LIN {X 0,Y 474.583,Z 139.364,A -85,B 0,C 180,E1 -7443.623,E2 -7443.623} C_VEL
LIN {X 0,Y 474.627,Z 139.367,A -85,B 0,C 180,E1 -7446.642,E2 -7446.642} C_VEL
LIN {X 0,Y 474.635,Z 139.36,A -85,B 0,C 180,E1 -7450.088,E2 -7450.088} C_VEL
LIN {X 0,Y 474.63,Z 139.358,A -85,B 0,C 180,E1 -7451.634,E2 -7451.634} C_VEL
LIN {X 0,Y 473.949,Z 139.45,A -85,B 0,C 180,E1 -7452.343,E2 -7452.343} C_VEL
LIN {X 0,Y 471.1,Z 139.8,A -85,B 0,C 180,E1 -7453.494,E2 -7453.494} C_VEL
LIN {X 0,Y 468.697,Z 140.106,A -85,B 0,C 180,E1 -7454.421,E2 -7454.421} C_VEL
LIN {X 0,Y 467.662,Z 140.228,A -85,B 0,C 180,E1 -7455.138,E2 -7455.138} C_VEL
LIN {X 0,Y 467.575,Z 140.237,A -85,B 0,C 180,E1 -7455.381,E2 -7455.381} C_VEL
LIN {X 0,Y 467.64,Z 140.231,A -85,B 0,C 180,E1 -7457.854,E2 -7457.854} C_VEL
LIN {X 0,Y 467.625,Z 140.231,A -85,B 0,C 180,E1 -7461.356,E2 -7461.356} C_VEL
LIN {X 0,Y 467.692,Z 140.228,A -85,B 0,C 180,E1 -7463.962,E2 -7463.962} C_VEL
LIN {X 0,Y 467.804,Z 140.212,A -85,B 0,C 180,E1 -7467.417,E2 -7467.417} C_VEL
LIN {X 0,Y 467.841,Z 140.213,A -85,B 0,C 180,E1 -7470,E2 -7470} C_VEL
LIN {X 0,Y 467.646,Z 140.35,A -85,B 0,C 180,E1 -7471.049,E2 -7471.049} C_VEL
LIN {X 0,Y 468.659,Z 146.382,A -85,B 0,C 180,E1 -7472.363,E2 -7472.363} C_VEL
LIN {X 0,Y 468.453,Z 159.385,A -85,B 0,C 180,E1 -7475.056,E2 -7475.056} C_VEL
LIN {X 0,Y 471.335,Z 174.004,A -85,B 0,C 180,E1 -7475.401,E2 -7475.401} C_VEL
LIN {X 0,Y 470.568,Z 266.04,A -85,B 0,C 180,E1 -7476.835,E2 -7476.835} C_VEL
LIN {X 0,Y 470.243,Z 278.777,A -85,B 0,C 180,E1 -7477.19,E2 -7477.19} C_VEL
LIN {X 0,Y 469.971,Z 291.673,A -85,B 0,C 180,E1 -7477.735,E2 -7477.735} C_VEL
LIN {X 0,Y 469.608,Z 303.175,A -85,B 0,C 180,E1 -7478.39,E2 -7478.39} C_VEL
LIN {X 0,Y 469.175,Z 313.348,A -85,B 0,C 180,E1 -7479.128,E2 -7479.128} C_VEL
LIN {X 0,Y 468.657,Z 324.539,A -85,B 0,C 180,E1 -7480.149,E2 -7480.149} C_VEL
LIN {X 0,Y 468.147,Z 334.312,A -85,B 0,C 180,E1 -7481.254,E2 -7481.254} C_VEL
LIN {X 0,Y 467.723,Z 342.539,A -85,B 0,C 180,E1 -7482.4,E2 -7482.4} C_VEL
LIN {X 0,Y 467.364,Z 350.081,A -85,B 0,C 180,E1 -7483.7,E2 -7483.7} C_VEL
LIN {X 0,Y 467.052,Z 357.038,A -85,B 0,C 180,E1 -7485.214,E2 -7485.214} C_VEL
LIN {X 0,Y 466.866,Z 361.993,A -85,B 0,C 180,E1 -7486.62,E2 -7486.62} C_VEL
LIN {X 0,Y 466.721,Z 365.558,A -85,B 0,C 180,E1 -7487.974,E2 -7487.974} C_VEL
LIN {X 0,Y 466.61,Z 368.078,A -85,B 0,C 180,E1 -7489.351,E2 -7489.351} C_VEL
LIN {X 0,Y 466.545,Z 369.678,A -85,B 0,C 180,E1 -7490.942,E2 -7490.942} C_VEL
LIN {X 0,Y 466.524,Z 370.029,A -85,B 0,C 180,E1 -7492.124,E2 -7492.124} C_VEL
LIN {X 0,Y 466.578,Z 369.644,A -85,B 0,C 180,E1 -7493.246,E2 -7493.246} C_VEL
LIN {X 0,Y 466.622,Z 367.819,A -85,B 0,C 180,E1 -7494.943,E2 -7494.943} C_VEL
LIN {X 0,Y 466.775,Z 365.039,A -85,B 0,C 180,E1 -7496.37,E2 -7496.37} C_VEL
LIN {X 0,Y 466.957,Z 361.004,A -85,B 0,C 180,E1 -7497.812,E2 -7497.812} C_VEL
LIN {X 0,Y 467.117,Z 355.698,A -85,B 0,C 180,E1 -7499.236,E2 -7499.236} C_VEL
LIN {X 0,Y 467.404,Z 349.728,A -85,B 0,C 180,E1 -7500.496,E2 -7500.496} C_VEL
LIN {X 0,Y 467.742,Z 342.532,A -85,B 0,C 180,E1 -7501.728,E2 -7501.728} C_VEL
LIN {X 0,Y 468.227,Z 333.765,A -85,B 0,C 180,E1 -7502.938,E2 -7502.938} C_VEL
LIN {X 0,Y 468.666,Z 323.643,A -85,B 0,C 180,E1 -7504.07,E2 -7504.07} C_VEL
LIN {X 0,Y 469.176,Z 313.829,A -85,B 0,C 180,E1 -7504.957,E2 -7504.957} C_VEL
LIN {X 0,Y 469.676,Z 302.364,A -85,B 0,C 180,E1 -7505.784,E2 -7505.784} C_VEL
LIN {X 0,Y 470.13,Z 290.08,A -85,B 0,C 180,E1 -7506.463,E2 -7506.463} C_VEL
LIN {X 0,Y 470.434,Z 277.293,A -85,B 0,C 180,E1 -7506.981,E2 -7506.981} C_VEL
LIN {X 0,Y 470.671,Z 264.549,A -85,B 0,C 180,E1 -7507.311,E2 -7507.311} C_VEL
LIN {X 0,Y 471.315,Z 173.329,A -85,B 0,C 180,E1 -7508.736,E2 -7508.736} C_VEL
LIN {X 0,Y 468.55,Z 159.48,A -85,B 0,C 180,E1 -7509.086,E2 -7509.086} C_VEL
LIN {X 0,Y 468.857,Z 147.777,A -85,B 0,C 180,E1 -7511.456,E2 -7511.456} C_VEL
LIN {X 0,Y 467.637,Z 140.236,A -85,B 0,C 180,E1 -7513.07,E2 -7513.07} C_VEL
LIN {X 0,Y 467.573,Z 140.242,A -85,B 0,C 180,E1 -7516.259,E2 -7516.259} C_VEL
LIN {X 0,Y 467.586,Z 140.24,A -85,B 0,C 180,E1 -7518.722,E2 -7518.722} C_VEL
LIN {X 0,Y 467.566,Z 140.248,A -85,B 0,C 180,E1 -7521.957,E2 -7521.957} C_VEL
LIN {X 0,Y 467.562,Z 140.244,A -85,B 0,C 180,E1 -7525.168,E2 -7525.168} C_VEL
LIN {X 0,Y 467.58,Z 140.238,A -85,B 0,C 180,E1 -7528.261,E2 -7528.261} C_VEL
LIN {X 0,Y 467.575,Z 140.243,A -85,B 0,C 180,E1 -7531.251,E2 -7531.251} C_VEL
LIN {X 0,Y 467.609,Z 140.236,A -85,B 0,C 180,E1 -7534.161,E2 -7534.161} C_VEL
LIN {X 0,Y 467.576,Z 140.243,A -85,B 0,C 180,E1 -7536.997,E2 -7536.997} C_VEL
LIN {X 0,Y 467.621,Z 140.234,A -85,B 0,C 180,E1 -7539.778,E2 -7539.778} C_VEL
LIN {X 0,Y 467.595,Z 140.237,A -85,B 0,C 180,E1 -7542.507,E2 -7542.507} C_VEL
LIN {X 0,Y 467.605,Z 140.238,A -85,B 0,C 180,E1 -7545.197,E2 -7545.197} C_VEL
LIN {X 0,Y 467.657,Z 140.227,A -85,B 0,C 180,E1 -7547.855,E2 -7547.855} C_VEL
LIN {X 0,Y 467.67,Z 140.224,A -85,B 0,C 180,E1 -7551.358,E2 -7551.358} C_VEL
LIN {X 0,Y 467.724,Z 140.22,A -85,B 0,C 180,E1 -7553.963,E2 -7553.963} C_VEL
LIN {X 0,Y 467.852,Z 140.201,A -85,B 0,C 180,E1 -7557.418,E2 -7557.418} C_VEL
LIN {X 0,Y 467.88,Z 140.2,A -85,B 0,C 180,E1 -7560.001,E2 -7560.001} C_VEL
LIN {X 0,Y 467.818,Z 140.211,A -85,B 0,C 180,E1 -7562.584,E2 -7562.584} C_VEL
LIN {X 0,Y 467.712,Z 140.219,A -85,B 0,C 180,E1 -7566.038,E2 -7566.038} C_VEL
LIN {X 0,Y 467.66,Z 140.228,A -85,B 0,C 180,E1 -7568.644,E2 -7568.644} C_VEL
LIN {X 0,Y 467.659,Z 140.231,A -85,B 0,C 180,E1 -7572.146,E2 -7572.146} C_VEL
LIN {X 0,Y 467.616,Z 140.236,A -85,B 0,C 180,E1 -7575.696,E2 -7575.696} C_VEL
LIN {X 0,Y 467.617,Z 140.235,A -85,B 0,C 180,E1 -7579.309,E2 -7579.309} C_VEL
LIN {X 0,Y 467.525,Z 140.246,A -85,B 0,C 180,E1 -7582.075,E2 -7582.075} C_VEL
LIN {X 0,Y 467.561,Z 140.24,A -85,B 0,C 180,E1 -7584.89,E2 -7584.89} C_VEL
LIN {X 0,Y 467.541,Z 140.247,A -85,B 0,C 180,E1 -7587.775,E2 -7587.775} C_VEL
LIN {X 0,Y 467.529,Z 140.243,A -85,B 0,C 180,E1 -7591.037,E2 -7591.037} C_VEL
LIN {X 0,Y 467.564,Z 140.237,A -85,B 0,C 180,E1 -7594.238,E2 -7594.238} C_VEL
LIN {X 0,Y 467.512,Z 140.251,A -85,B 0,C 180,E1 -7597.18,E2 -7597.18} C_VEL
LIN {X 0,Y 467.519,Z 140.247,A -85,B 0,C 180,E1 -7600.271,E2 -7600.271} C_VEL
LIN {X 0,Y 467.518,Z 140.25,A -85,B 0,C 180,E1 -7602.569,E2 -7602.569} C_VEL
LIN {X 0,Y 467.564,Z 140.249,A -85,B 0,C 180,E1 -7605.052,E2 -7605.052} C_VEL
LIN {X 0,Y 467.562,Z 140.248,A -85,B 0,C 180,E1 -7608.726,E2 -7608.726} C_VEL
LIN {X 0,Y 467.554,Z 140.243,A -85,B 0,C 180,E1 -7611.954,E2 -7611.954} C_VEL
LIN {X 0,Y 467.557,Z 140.242,A -85,B 0,C 180,E1 -7615.167,E2 -7615.167} C_VEL
LIN {X 0,Y 467.58,Z 140.242,A -85,B 0,C 180,E1 -7618.26,E2 -7618.26} C_VEL
LIN {X 0,Y 467.547,Z 140.245,A -85,B 0,C 180,E1 -7621.248,E2 -7621.248} C_VEL
LIN {X 0,Y 467.602,Z 140.403,A -85,B 0,C 180,E1 -7624.04,E2 -7624.04} C_VEL
LIN {X 0,Y 469.779,Z 151.706,A -85,B 0,C 180,E1 -7626.176,E2 -7626.176} C_VEL
LIN {X 0,Y 469.174,Z 167.509,A -85,B 0,C 180,E1 -7628.93,E2 -7628.93} C_VEL
LIN {X 0,Y 468.445,Z 185.894,A -85,B 0,C 180,E1 -7632.088,E2 -7632.088} C_VEL
LIN {X 0,Y 468.286,Z 190.998,A -85,B 0,C 180,E1 -7632.958,E2 -7632.958} C_VEL
LIN {X 0,Y 471.16,Z 210.073,A -85,B 0,C 180,E1 -7633.369,E2 -7633.369} C_VEL
LIN {X 0,Y 470.551,Z 299.268,A -85,B 0,C 180,E1 -7634.765,E2 -7634.765} C_VEL
LIN {X 0,Y 470.212,Z 311.843,A -85,B 0,C 180,E1 -7635.114,E2 -7635.114} C_VEL
LIN {X 0,Y 469.706,Z 324.813,A -85,B 0,C 180,E1 -7635.652,E2 -7635.652} C_VEL
LIN {X 0,Y 469.186,Z 337.139,A -85,B 0,C 180,E1 -7636.354,E2 -7636.354} C_VEL
LIN {X 0,Y 468.715,Z 347.709,A -85,B 0,C 180,E1 -7637.132,E2 -7637.132} C_VEL
LIN {X 0,Y 468.201,Z 359.257,A -85,B 0,C 180,E1 -7638.199,E2 -7638.199} C_VEL
LIN {X 0,Y 467.748,Z 367.831,A -85,B 0,C 180,E1 -7639.175,E2 -7639.175} C_VEL
LIN {X 0,Y 467.399,Z 375.747,A -85,B 0,C 180,E1 -7640.261,E2 -7640.261} C_VEL
LIN {X 0,Y 467.089,Z 383.481,A -85,B 0,C 180,E1 -7641.564,E2 -7641.564} C_VEL
LIN {X 0,Y 466.831,Z 390.612,A -85,B 0,C 180,E1 -7643.083,E2 -7643.083} C_VEL
LIN {X 0,Y 466.73,Z 395.361,A -85,B 0,C 180,E1 -7644.383,E2 -7644.383} C_VEL
LIN {X 0,Y 466.646,Z 398.989,A -85,B 0,C 180,E1 -7645.682,E2 -7645.682} C_VEL
LIN {X 0,Y 466.69,Z 400.865,A -85,B 0,C 180,E1 -7646.547,E2 -7646.547} C_VEL
LIN {X 0,Y 466.663,Z 402.269,A -85,B 0,C 180,E1 -7647.411,E2 -7647.411} C_VEL
LIN {X 0,Y 466.623,Z 403.887,A -85,B 0,C 180,E1 -7649.137,E2 -7649.137} C_VEL
LIN {X 0,Y 466.605,Z 404.106,A -85,B 0,C 180,E1 -7650,E2 -7650} C_VEL
LIN {X 0,Y 466.623,Z 403.89,A -85,B 0,C 180,E1 -7650.863,E2 -7650.863} C_VEL
LIN {X 0,Y 466.663,Z 402.286,A -85,B 0,C 180,E1 -7652.59,E2 -7652.59} C_VEL
LIN {X 0,Y 466.69,Z 400.884,A -85,B 0,C 180,E1 -7653.454,E2 -7653.454} C_VEL
LIN {X 0,Y 466.687,Z 397.935,A -85,B 0,C 180,E1 -7654.751,E2 -7654.751} C_VEL
LIN {X 0,Y 466.742,Z 393.941,A -85,B 0,C 180,E1 -7656.051,E2 -7656.051} C_VEL
LIN {X 0,Y 466.94,Z 387.795,A -85,B 0,C 180,E1 -7657.568,E2 -7657.568} C_VEL
LIN {X 0,Y 467.157,Z 381.082,A -85,B 0,C 180,E1 -7658.871,E2 -7658.871} C_VEL
LIN {X 0,Y 467.487,Z 372.755,A -85,B 0,C 180,E1 -7660.175,E2 -7660.175} C_VEL
LIN {X 0,Y 467.938,Z 364.206,A -85,B 0,C 180,E1 -7661.259,E2 -7661.259} C_VEL
LIN {X 0,Y 468.417,Z 354.192,A -85,B 0,C 180,E1 -7662.295,E2 -7662.295} C_VEL
LIN {X 0,Y 468.867,Z 343.19,A -85,B 0,C 180,E1 -7663.214,E2 -7663.214} C_VEL
LIN {X 0,Y 469.4,Z 331.709,A -85,B 0,C 180,E1 -7663.971,E2 -7663.971} C_VEL
LIN {X 0,Y 469.898,Z 319.834,A -85,B 0,C 180,E1 -7664.564,E2 -7664.564} C_VEL
LIN {X 0,Y 470.318,Z 307.042,A -85,B 0,C 180,E1 -7665.021,E2 -7665.021} C_VEL
LIN {X 0,Y 470.601,Z 293.776,A -85,B 0,C 180,E1 -7665.317,E2 -7665.317} C_VEL
LIN {X 0,Y 471.015,Z 209.408,A -85,B 0,C 180,E1 -7666.623,E2 -7666.623} C_VEL
LIN {X 0,Y 468.255,Z 191.282,A -85,B 0,C 180,E1 -7667.019,E2 -7667.019} C_VEL
LIN {X 0,Y 468.913,Z 174.317,A -85,B 0,C 180,E1 -7669.937,E2 -7669.937} C_VEL
LIN {X 0,Y 469.668,Z 158.629,A -85,B 0,C 180,E1 -7672.664,E2 -7672.664} C_VEL
LIN {X 0,Y 469.843,Z 152.075,A -85,B 0,C 180,E1 -7673.821,E2 -7673.821} C_VEL
LIN {X 0,Y 467.567,Z 140.242,A -85,B 0,C 180,E1 -7676.082,E2 -7676.082} C_VEL
LIN {X 0,Y 467.554,Z 140.247,A -85,B 0,C 180,E1 -7679.328,E2 -7679.328} C_VEL
LIN {X 0,Y 467.582,Z 140.244,A -85,B 0,C 180,E1 -7681.741,E2 -7681.741} C_VEL
LIN {X 0,Y 467.56,Z 140.24,A -85,B 0,C 180,E1 -7684.833,E2 -7684.833} C_VEL
LIN {X 0,Y 467.565,Z 140.24,A -85,B 0,C 180,E1 -7688.045,E2 -7688.045} C_VEL
LIN {X 0,Y 467.565,Z 140.245,A -85,B 0,C 180,E1 -7691.274,E2 -7691.274} C_VEL
LIN {X 0,Y 467.57,Z 140.241,A -85,B 0,C 180,E1 -7694.948,E2 -7694.948} C_VEL
LIN {X 0,Y 467.563,Z 140.24,A -85,B 0,C 180,E1 -7698.595,E2 -7698.595} C_VEL
LIN {X 0,Y 467.561,Z 140.244,A -85,B 0,C 180,E1 -7701.41,E2 -7701.41} C_VEL
LIN {X 0,Y 467.562,Z 140.239,A -85,B 0,C 180,E1 -7704.261,E2 -7704.261} C_VEL
LIN {X 0,Y 467.578,Z 140.241,A -85,B 0,C 180,E1 -7707.323,E2 -7707.323} C_VEL
LIN {X 0,Y 467.551,Z 140.245,A -85,B 0,C 180,E1 -7710.673,E2 -7710.673} C_VEL
LIN {X 0,Y 467.556,Z 140.243,A -85,B 0,C 180,E1 -7713.195,E2 -7713.195} C_VEL
LIN {X 0,Y 467.594,Z 140.239,A -85,B 0,C 180,E1 -7716.469,E2 -7716.469} C_VEL
LIN {X 0,Y 467.616,Z 140.232,A -85,B 0,C 180,E1 -7719.776,E2 -7719.776} C_VEL
LIN {X 0,Y 467.568,Z 140.244,A -85,B 0,C 180,E1 -7722.505,E2 -7722.505} C_VEL
LIN {X 0,Y 467.595,Z 140.236,A -85,B 0,C 180,E1 -7725.195,E2 -7725.195} C_VEL
LIN {X 0,Y 467.662,Z 140.227,A -85,B 0,C 180,E1 -7727.854,E2 -7727.854} C_VEL
LIN {X 0,Y 467.641,Z 140.229,A -85,B 0,C 180,E1 -7731.356,E2 -7731.356} C_VEL
LIN {X 0,Y 467.706,Z 140.224,A -85,B 0,C 180,E1 -7733.961,E2 -7733.961} C_VEL
LIN {X 0,Y 467.817,Z 140.207,A -85,B 0,C 180,E1 -7737.416,E2 -7737.416} C_VEL
LIN {X 0,Y 467.853,Z 140.208,A -85,B 0,C 180,E1 -7739.999,E2 -7739.999} C_VEL
LIN {X 0,Y 467.816,Z 140.21,A -85,B 0,C 180,E1 -7742.582,E2 -7742.582} C_VEL
LIN {X 0,Y 467.704,Z 140.229,A -85,B 0,C 180,E1 -7746.037,E2 -7746.037} C_VEL
LIN {X 0,Y 467.636,Z 140.231,A -85,B 0,C 180,E1 -7748.643,E2 -7748.643} C_VEL
LIN {X 0,Y 467.651,Z 140.233,A -85,B 0,C 180,E1 -7752.145,E2 -7752.145} C_VEL
LIN {X 0,Y 467.607,Z 140.239,A -85,B 0,C 180,E1 -7755.695,E2 -7755.695} C_VEL
LIN {X 0,Y 467.574,Z 140.237,A -85,B 0,C 180,E1 -7758.747,E2 -7758.747} C_VEL
LIN {X 0,Y 467.559,Z 140.242,A -85,B 0,C 180,E1 -7761.26,E2 -7761.26} C_VEL
LIN {X 0,Y 467.555,Z 140.244,A -85,B 0,C 180,E1 -7763.943,E2 -7763.943} C_VEL
LIN {X 0,Y 467.534,Z 140.243,A -85,B 0,C 180,E1 -7766.804,E2 -7766.804} C_VEL
LIN {X 0,Y 467.533,Z 140.248,A -85,B 0,C 180,E1 -7769.739,E2 -7769.739} C_VEL
LIN {X 0,Y 467.572,Z 140.238,A -85,B 0,C 180,E1 -7772.758,E2 -7772.758} C_VEL
LIN {X 0,Y 467.547,Z 140.243,A -85,B 0,C 180,E1 -7775.889,E2 -7775.889} C_VEL
LIN {X 0,Y 467.542,Z 140.248,A -85,B 0,C 180,E1 -7779.148,E2 -7779.148} C_VEL
LIN {X 0,Y 467.555,Z 140.245,A -85,B 0,C 180,E1 -7781.404,E2 -7781.404} C_VEL
LIN {X 0,Y 467.562,Z 140.246,A -85,B 0,C 180,E1 -7785.051,E2 -7785.051} C_VEL
LIN {X 0,Y 467.556,Z 140.243,A -85,B 0,C 180,E1 -7788.725,E2 -7788.725} C_VEL
LIN {X 0,Y 467.556,Z 140.24,A -85,B 0,C 180,E1 -7791.954,E2 -7791.954} C_VEL
LIN {X 0,Y 467.549,Z 140.245,A -85,B 0,C 180,E1 -7795.166,E2 -7795.166} C_VEL
LIN {X 0,Y 467.551,Z 140.242,A -85,B 0,C 180,E1 -7798.257,E2 -7798.257} C_VEL
LIN {X 0,Y 467.534,Z 140.245,A -85,B 0,C 180,E1 -7801.247,E2 -7801.247} C_VEL
LIN {X 0,Y 467.571,Z 140.242,A -85,B 0,C 180,E1 -7804.4,E2 -7804.4} C_VEL
LIN {X 0,Y 467.561,Z 140.242,A -85,B 0,C 180,E1 -7806.995,E2 -7806.995} C_VEL
LIN {X 0,Y 467.603,Z 140.234,A -85,B 0,C 180,E1 -7809.776,E2 -7809.776} C_VEL
LIN {X 0,Y 467.554,Z 140.248,A -85,B 0,C 180,E1 -7812.504,E2 -7812.504} C_VEL
LIN {X 0,Y 467.575,Z 140.237,A -85,B 0,C 180,E1 -7815.381,E2 -7815.381} C_VEL
LIN {X 0,Y 466.905,Z 140.327,A -85,B 0,C 180,E1 -7816.1,E2 -7816.1} C_VEL
LIN {X 0,Y 464.062,Z 140.677,A -85,B 0,C 180,E1 -7817.269,E2 -7817.269} C_VEL
LIN {X 0,Y 461.661,Z 140.98,A -85,B 0,C 180,E1 -7818.211,E2 -7818.211} C_VEL
LIN {X 0,Y 460.628,Z 141.104,A -85,B 0,C 180,E1 -7818.939,E2 -7818.939} C_VEL
LIN {X 0,Y 460.542,Z 141.113,A -85,B 0,C 180,E1 -7819.185,E2 -7819.185} C_VEL
LIN {X 0,Y 460.654,Z 141.103,A -85,B 0,C 180,E1 -7822.594,E2 -7822.594} C_VEL
LIN {X 0,Y 460.664,Z 141.1,A -85,B 0,C 180,E1 -7824.748,E2 -7824.748} C_VEL
LIN {X 0,Y 460.748,Z 141.091,A -85,B 0,C 180,E1 -7827.377,E2 -7827.377} C_VEL
LIN {X 0,Y 460.81,Z 141.088,A -85,B 0,C 180,E1 -7830,E2 -7830} C_VEL
LIN {X 0,Y 460.586,Z 141.229,A -85,B 0,C 180,E1 -7830.874,E2 -7830.874} C_VEL
LIN {X 0,Y 461.719,Z 148.149,A -85,B 0,C 180,E1 -7832.399,E2 -7832.399} C_VEL
LIN {X 0,Y 461.482,Z 159.661,A -85,B 0,C 180,E1 -7834.805,E2 -7834.805} C_VEL
LIN {X 0,Y 464.575,Z 175.741,A -85,B 0,C 180,E1 -7835.18,E2 -7835.18} C_VEL
LIN {X 0,Y 463.695,Z 267.36,A -85,B 0,C 180,E1 -7836.636,E2 -7836.636} C_VEL
LIN {X 0,Y 463.354,Z 280.48,A -85,B 0,C 180,E1 -7837.024,E2 -7837.024} C_VEL
LIN {X 0,Y 463.065,Z 293,A -85,B 0,C 180,E1 -7837.576,E2 -7837.576} C_VEL
LIN {X 0,Y 462.636,Z 305.012,A -85,B 0,C 180,E1 -7838.298,E2 -7838.298} C_VEL
LIN {X 0,Y 462.145,Z 316.016,A -85,B 0,C 180,E1 -7839.144,E2 -7839.144} C_VEL
LIN {X 0,Y 461.612,Z 326.922,A -85,B 0,C 180,E1 -7840.194,E2 -7840.194} C_VEL
LIN {X 0,Y 461.021,Z 337.089,A -85,B 0,C 180,E1 -7841.43,E2 -7841.43} C_VEL
LIN {X 0,Y 460.58,Z 345.739,A -85,B 0,C 180,E1 -7842.738,E2 -7842.738} C_VEL
LIN {X 0,Y 460.191,Z 353.114,A -85,B 0,C 180,E1 -7844.143,E2 -7844.143} C_VEL
LIN {X 0,Y 459.937,Z 359.517,A -85,B 0,C 180,E1 -7845.71,E2 -7845.71} C_VEL
LIN {X 0,Y 459.743,Z 363.224,A -85,B 0,C 180,E1 -7846.885,E2 -7846.885} C_VEL
LIN {X 0,Y 459.67,Z 365.569,A -85,B 0,C 180,E1 -7847.805,E2 -7847.805} C_VEL
LIN {X 0,Y 459.564,Z 367.404,A -85,B 0,C 180,E1 -7848.732,E2 -7848.732} C_VEL
LIN {X 0,Y 459.511,Z 368.783,A -85,B 0,C 180,E1 -7849.662,E2 -7849.662} C_VEL
LIN {X 0,Y 459.453,Z 370.021,A -85,B 0,C 180,E1 -7851.082,E2 -7851.082} C_VEL
LIN {X 0,Y 459.44,Z 370.226,A -85,B 0,C 180,E1 -7852.484,E2 -7852.484} C_VEL
LIN {X 0,Y 459.482,Z 369.814,A -85,B 0,C 180,E1 -7853.433,E2 -7853.433} C_VEL
LIN {X 0,Y 459.511,Z 368.885,A -85,B 0,C 180,E1 -7854.39,E2 -7854.39} C_VEL
LIN {X 0,Y 459.608,Z 367.149,A -85,B 0,C 180,E1 -7855.555,E2 -7855.555} C_VEL
LIN {X 0,Y 459.755,Z 364.424,A -85,B 0,C 180,E1 -7856.805,E2 -7856.805} C_VEL
LIN {X 0,Y 459.907,Z 360.061,A -85,B 0,C 180,E1 -7858.276,E2 -7858.276} C_VEL
LIN {X 0,Y 460.194,Z 353.89,A -85,B 0,C 180,E1 -7859.823,E2 -7859.823} C_VEL
LIN {X 0,Y 460.555,Z 346.372,A -85,B 0,C 180,E1 -7861.292,E2 -7861.292} C_VEL
LIN {X 0,Y 460.975,Z 338.559,A -85,B 0,C 180,E1 -7862.507,E2 -7862.507} C_VEL
LIN {X 0,Y 461.445,Z 329.596,A -85,B 0,C 180,E1 -7863.642,E2 -7863.642} C_VEL
LIN {X 0,Y 462.012,Z 318.546,A -85,B 0,C 180,E1 -7864.773,E2 -7864.773} C_VEL
LIN {X 0,Y 462.563,Z 307.476,A -85,B 0,C 180,E1 -7865.666,E2 -7865.666} C_VEL
LIN {X 0,Y 463.084,Z 296.331,A -85,B 0,C 180,E1 -7866.372,E2 -7866.372} C_VEL
LIN {X 0,Y 463.454,Z 283.37,A -85,B 0,C 180,E1 -7866.996,E2 -7866.996} C_VEL
LIN {X 0,Y 463.718,Z 270.876,A -85,B 0,C 180,E1 -7867.408,E2 -7867.408} C_VEL
LIN {X 0,Y 463.942,Z 254.464,A -85,B 0,C 180,E1 -7867.718,E2 -7867.718} C_VEL
LIN {X 0,Y 464.625,Z 174.638,A -85,B 0,C 180,E1 -7868.972,E2 -7868.972} C_VEL
LIN {X 0,Y 461.627,Z 159.77,A -85,B 0,C 180,E1 -7869.35,E2 -7869.35} C_VEL
LIN {X 0,Y 461.894,Z 149.544,A -85,B 0,C 180,E1 -7871.443,E2 -7871.443} C_VEL
LIN {X 0,Y 461.043,Z 143.561,A -85,B 0,C 180,E1 -7872.725,E2 -7872.725} C_VEL
LIN {X 0,Y 460.581,Z 141.115,A -85,B 0,C 180,E1 -7873.273,E2 -7873.273} C_VEL
LIN {X 0,Y 460.521,Z 141.118,A -85,B 0,C 180,E1 -7876.628,E2 -7876.628} C_VEL
LIN {X 0,Y 460.556,Z 141.123,A -85,B 0,C 180,E1 -7879.729,E2 -7879.729} C_VEL
LIN {X 0,Y 460.524,Z 141.121,A -85,B 0,C 180,E1 -7882.52,E2 -7882.52} C_VEL
LIN {X 0,Y 460.544,Z 141.122,A -85,B 0,C 180,E1 -7885.625,E2 -7885.625} C_VEL
LIN {X 0,Y 460.535,Z 141.116,A -85,B 0,C 180,E1 -7888.745,E2 -7888.745} C_VEL
LIN {X 0,Y 460.58,Z 141.11,A -85,B 0,C 180,E1 -7892.255,E2 -7892.255} C_VEL
LIN {X 0,Y 460.558,Z 141.116,A -85,B 0,C 180,E1 -7894.706,E2 -7894.706} C_VEL
LIN {X 0,Y 460.51,Z 141.123,A -85,B 0,C 180,E1 -7897.572,E2 -7897.572} C_VEL
LIN {X 0,Y 460.567,Z 141.112,A -85,B 0,C 180,E1 -7900.385,E2 -7900.385} C_VEL
LIN {X 0,Y 460.604,Z 141.107,A -85,B 0,C 180,E1 -7904.06,E2 -7904.06} C_VEL
LIN {X 0,Y 460.61,Z 141.105,A -85,B 0,C 180,E1 -7907.667,E2 -7907.667} C_VEL
LIN {X 0,Y 460.62,Z 141.103,A -85,B 0,C 180,E1 -7911.224,E2 -7911.224} C_VEL
LIN {X 0,Y 460.688,Z 141.096,A -85,B 0,C 180,E1 -7913.871,E2 -7913.871} C_VEL
LIN {X 0,Y 460.793,Z 141.081,A -85,B 0,C 180,E1 -7917.378,E2 -7917.378} C_VEL
LIN {X 0,Y 460.85,Z 141.075,A -85,B 0,C 180,E1 -7920.001,E2 -7920.001} C_VEL
LIN {X 0,Y 460.761,Z 141.089,A -85,B 0,C 180,E1 -7922.623,E2 -7922.623} C_VEL
LIN {X 0,Y 460.677,Z 141.096,A -85,B 0,C 180,E1 -7926.131,E2 -7926.131} C_VEL
LIN {X 0,Y 460.612,Z 141.105,A -85,B 0,C 180,E1 -7928.777,E2 -7928.777} C_VEL
LIN {X 0,Y 460.612,Z 141.109,A -85,B 0,C 180,E1 -7932.335,E2 -7932.335} C_VEL
LIN {X 0,Y 460.56,Z 141.112,A -85,B 0,C 180,E1 -7935.979,E2 -7935.979} C_VEL
LIN {X 0,Y 460.562,Z 141.118,A -85,B 0,C 180,E1 -7939.616,E2 -7939.616} C_VEL
LIN {X 0,Y 460.497,Z 141.119,A -85,B 0,C 180,E1 -7942.43,E2 -7942.43} C_VEL
LIN {X 0,Y 460.537,Z 141.115,A -85,B 0,C 180,E1 -7945.794,E2 -7945.794} C_VEL
LIN {X 0,Y 460.498,Z 141.12,A -85,B 0,C 180,E1 -7948.237,E2 -7948.237} C_VEL
LIN {X 0,Y 460.498,Z 141.122,A -85,B 0,C 180,E1 -7951.278,E2 -7951.278} C_VEL
LIN {X 0,Y 460.509,Z 141.116,A -85,B 0,C 180,E1 -7954.501,E2 -7954.501} C_VEL
LIN {X 0,Y 460.481,Z 141.122,A -85,B 0,C 180,E1 -7957.626,E2 -7957.626} C_VEL
LIN {X 0,Y 460.501,Z 141.125,A -85,B 0,C 180,E1 -7961.015,E2 -7961.015} C_VEL
LIN {X 0,Y 460.512,Z 141.122,A -85,B 0,C 180,E1 -7964.59,E2 -7964.59} C_VEL
LIN {X 0,Y 460.476,Z 141.126,A -85,B 0,C 180,E1 -7967.813,E2 -7967.813} C_VEL
LIN {X 0,Y 460.513,Z 141.122,A -85,B 0,C 180,E1 -7970.136,E2 -7970.136} C_VEL
LIN {X 0,Y 460.472,Z 141.121,A -85,B 0,C 180,E1 -7973.47,E2 -7973.47} C_VEL
LIN {X 0,Y 460.519,Z 141.122,A -85,B 0,C 180,E1 -7976.674,E2 -7976.674} C_VEL
LIN {X 0,Y 460.507,Z 141.122,A -85,B 0,C 180,E1 -7979.76,E2 -7979.76} C_VEL
LIN {X 0,Y 460.495,Z 141.125,A -85,B 0,C 180,E1 -7982.751,E2 -7982.751} C_VEL
LIN {X 0,Y 460.537,Z 141.176,A -85,B 0,C 180,E1 -7983.797,E2 -7983.797} C_VEL
LIN {X 0,Y 462.784,Z 152.783,A -85,B 0,C 180,E1 -7986.032,E2 -7986.032} C_VEL
LIN {X 0,Y 462.56,Z 162.007,A -85,B 0,C 180,E1 -7987.676,E2 -7987.676} C_VEL
LIN {X 0,Y 461.696,Z 181.046,A -85,B 0,C 180,E1 -7991.008,E2 -7991.008} C_VEL
LIN {X 0,Y 461.353,Z 190.976,A -85,B 0,C 180,E1 -7992.694,E2 -7992.694} C_VEL
LIN {X 0,Y 464.375,Z 211.895,A -85,B 0,C 180,E1 -7993.147,E2 -7993.147} C_VEL
LIN {X 0,Y 463.709,Z 299.137,A -85,B 0,C 180,E1 -7994.535,E2 -7994.535} C_VEL
LIN {X 0,Y 463.332,Z 311.658,A -85,B 0,C 180,E1 -7994.888,E2 -7994.888} C_VEL
LIN {X 0,Y 462.826,Z 324.606,A -85,B 0,C 180,E1 -7995.434,E2 -7995.434} C_VEL
LIN {X 0,Y 462.277,Z 336.914,A -85,B 0,C 180,E1 -7996.146,E2 -7996.146} C_VEL
LIN {X 0,Y 461.768,Z 347.352,A -85,B 0,C 180,E1 -7996.924,E2 -7996.924} C_VEL
LIN {X 0,Y 461.269,Z 357.945,A -85,B 0,C 180,E1 -7997.907,E2 -7997.907} C_VEL
LIN {X 0,Y 460.76,Z 367.589,A -85,B 0,C 180,E1 -7999.009,E2 -7999.009} C_VEL
LIN {X 0,Y 460.364,Z 375.499,A -85,B 0,C 180,E1 -8000.111,E2 -8000.111} C_VEL
LIN {X 0,Y 460.028,Z 383.229,A -85,B 0,C 180,E1 -8001.434,E2 -8001.434} C_VEL
LIN {X 0,Y 459.746,Z 390.358,A -85,B 0,C 180,E1 -8002.976,E2 -8002.976} C_VEL
LIN {X 0,Y 459.63,Z 395.105,A -85,B 0,C 180,E1 -8004.296,E2 -8004.296} C_VEL
LIN {X 0,Y 459.563,Z 398.734,A -85,B 0,C 180,E1 -8005.615,E2 -8005.615} C_VEL
LIN {X 0,Y 459.585,Z 400.608,A -85,B 0,C 180,E1 -8006.493,E2 -8006.493} C_VEL
LIN {X 0,Y 459.585,Z 402.013,A -85,B 0,C 180,E1 -8007.371,E2 -8007.371} C_VEL
LIN {X 0,Y 459.556,Z 403.63,A -85,B 0,C 180,E1 -8009.124,E2 -8009.124} C_VEL
LIN {X 0,Y 459.537,Z 403.847,A -85,B 0,C 180,E1 -8010,E2 -8010} C_VEL
LIN {X 0,Y 459.556,Z 403.631,A -85,B 0,C 180,E1 -8010.876,E2 -8010.876} C_VEL
LIN {X 0,Y 459.585,Z 402.024,A -85,B 0,C 180,E1 -8012.63,E2 -8012.63} C_VEL
LIN {X 0,Y 459.585,Z 400.619,A -85,B 0,C 180,E1 -8013.507,E2 -8013.507} C_VEL
LIN {X 0,Y 459.615,Z 397.668,A -85,B 0,C 180,E1 -8014.825,E2 -8014.825} C_VEL
LIN {X 0,Y 459.694,Z 392.72,A -85,B 0,C 180,E1 -8016.407,E2 -8016.407} C_VEL
LIN {X 0,Y 459.883,Z 386.503,A -85,B 0,C 180,E1 -8017.906,E2 -8017.906} C_VEL
LIN {X 0,Y 460.161,Z 379.559,A -85,B 0,C 180,E1 -8019.228,E2 -8019.228} C_VEL
LIN {X 0,Y 460.455,Z 372.465,A -85,B 0,C 180,E1 -8020.332,E2 -8020.332} C_VEL
LIN {X 0,Y 460.933,Z 363.904,A -85,B 0,C 180,E1 -8021.433,E2 -8021.433} C_VEL
LIN {X 0,Y 461.436,Z 354.11,A -85,B 0,C 180,E1 -8022.462,E2 -8022.462} C_VEL
LIN {X 0,Y 461.928,Z 342.861,A -85,B 0,C 180,E1 -8023.416,E2 -8023.416} C_VEL
LIN {X 0,Y 462.504,Z 331.355,A -85,B 0,C 180,E1 -8024.184,E2 -8024.184} C_VEL
LIN {X 0,Y 463.021,Z 319.438,A -85,B 0,C 180,E1 -8024.785,E2 -8024.785} C_VEL
LIN {X 0,Y 463.464,Z 306.587,A -85,B 0,C 180,E1 -8025.249,E2 -8025.249} C_VEL
LIN {X 0,Y 463.734,Z 293.142,A -85,B 0,C 180,E1 -8025.549,E2 -8025.549} C_VEL
LIN {X 0,Y 464.278,Z 210.823,A -85,B 0,C 180,E1 -8026.84,E2 -8026.84} C_VEL
LIN {X 0,Y 461.326,Z 190.949,A -85,B 0,C 180,E1 -8027.292,E2 -8027.292} C_VEL
LIN {X 0,Y 461.986,Z 174.037,A -85,B 0,C 180,E1 -8030.248,E2 -8030.248} C_VEL
LIN {X 0,Y 462.712,Z 159.656,A -85,B 0,C 180,E1 -8032.788,E2 -8032.788} C_VEL
LIN {X 0,Y 462.867,Z 153.105,A -85,B 0,C 180,E1 -8033.964,E2 -8033.964} C_VEL
LIN {X 0,Y 460.531,Z 141.12,A -85,B 0,C 180,E1 -8036.298,E2 -8036.298} C_VEL
LIN {X 0,Y 460.521,Z 141.124,A -85,B 0,C 180,E1 -8039.555,E2 -8039.555} C_VEL
LIN {X 0,Y 460.529,Z 141.117,A -85,B 0,C 180,E1 -8042.285,E2 -8042.285} C_VEL
LIN {X 0,Y 460.51,Z 141.124,A -85,B 0,C 180,E1 -8045.446,E2 -8045.446} C_VEL
LIN {X 0,Y 460.508,Z 141.119,A -85,B 0,C 180,E1 -8048.891,E2 -8048.891} C_VEL
LIN {X 0,Y 460.506,Z 141.123,A -85,B 0,C 180,E1 -8051.598,E2 -8051.598} C_VEL
LIN {X 0,Y 460.516,Z 141.117,A -85,B 0,C 180,E1 -8054.589,E2 -8054.589} C_VEL
LIN {X 0,Y 460.48,Z 141.123,A -85,B 0,C 180,E1 -8057.813,E2 -8057.813} C_VEL
LIN {X 0,Y 460.517,Z 141.116,A -85,B 0,C 180,E1 -8060.135,E2 -8060.135} C_VEL
LIN {X 0,Y 460.477,Z 141.125,A -85,B 0,C 180,E1 -8063.47,E2 -8063.47} C_VEL
LIN {X 0,Y 460.521,Z 141.119,A -85,B 0,C 180,E1 -8066.674,E2 -8066.674} C_VEL
LIN {X 0,Y 460.502,Z 141.119,A -85,B 0,C 180,E1 -8069.759,E2 -8069.759} C_VEL
LIN {X 0,Y 460.517,Z 141.123,A -85,B 0,C 180,E1 -8072.752,E2 -8072.752} C_VEL
LIN {X 0,Y 460.522,Z 141.116,A -85,B 0,C 180,E1 -8075.666,E2 -8075.666} C_VEL
LIN {X 0,Y 460.524,Z 141.122,A -85,B 0,C 180,E1 -8078.579,E2 -8078.579} C_VEL
LIN {X 0,Y 460.587,Z 141.109,A -85,B 0,C 180,E1 -8081.31,E2 -8081.31} C_VEL
LIN {X 0,Y 460.552,Z 141.115,A -85,B 0,C 180,E1 -8084.964,E2 -8084.964} C_VEL
LIN {X 0,Y 460.614,Z 141.112,A -85,B 0,C 180,E1 -8088.559,E2 -8088.559} C_VEL
LIN {X 0,Y 460.599,Z 141.107,A -85,B 0,C 180,E1 -8091.223,E2 -8091.223} C_VEL
LIN {X 0,Y 460.672,Z 141.099,A -85,B 0,C 180,E1 -8093.869,E2 -8093.869} C_VEL
LIN {X 0,Y 460.761,Z 141.086,A -85,B 0,C 180,E1 -8097.377,E2 -8097.377} C_VEL
LIN {X 0,Y 460.823,Z 141.083,A -85,B 0,C 180,E1 -8099.999,E2 -8099.999} C_VEL
LIN {X 0,Y 460.759,Z 141.089,A -85,B 0,C 180,E1 -8102.622,E2 -8102.622} C_VEL
LIN {X 0,Y 460.67,Z 141.105,A -85,B 0,C 180,E1 -8106.13,E2 -8106.13} C_VEL
LIN {X 0,Y 460.591,Z 141.108,A -85,B 0,C 180,E1 -8108.776,E2 -8108.776} C_VEL
LIN {X 0,Y 460.6,Z 141.108,A -85,B 0,C 180,E1 -8112.434,E2 -8112.434} C_VEL
LIN {X 0,Y 460.559,Z 141.117,A -85,B 0,C 180,E1 -8115.977,E2 -8115.977} C_VEL
LIN {X 0,Y 460.532,Z 141.115,A -85,B 0,C 180,E1 -8118.886,E2 -8118.886} C_VEL
LIN {X 0,Y 460.51,Z 141.122,A -85,B 0,C 180,E1 -8121.485,E2 -8121.485} C_VEL
LIN {X 0,Y 460.517,Z 141.117,A -85,B 0,C 180,E1 -8124.333,E2 -8124.333} C_VEL
LIN {X 0,Y 460.49,Z 141.124,A -85,B 0,C 180,E1 -8127.248,E2 -8127.248} C_VEL
LIN {X 0,Y 460.495,Z 141.12,A -85,B 0,C 180,E1 -8130.24,E2 -8130.24} C_VEL
LIN {X 0,Y 460.515,Z 141.124,A -85,B 0,C 180,E1 -8133.325,E2 -8133.325} C_VEL
LIN {X 0,Y 460.468,Z 141.123,A -85,B 0,C 180,E1 -8136.529,E2 -8136.529} C_VEL
LIN {X 0,Y 460.508,Z 141.119,A -85,B 0,C 180,E1 -8139.864,E2 -8139.864} C_VEL
LIN {X 0,Y 460.459,Z 141.128,A -85,B 0,C 180,E1 -8142.892,E2 -8142.892} C_VEL
LIN {X 0,Y 460.499,Z 141.119,A -85,B 0,C 180,E1 -8145.831,E2 -8145.831} C_VEL
LIN {X 0,Y 460.51,Z 141.125,A -85,B 0,C 180,E1 -8148.986,E2 -8148.986} C_VEL
LIN {X 0,Y 460.509,Z 141.122,A -85,B 0,C 180,E1 -8151.265,E2 -8151.265} C_VEL
LIN {X 0,Y 460.5,Z 141.122,A -85,B 0,C 180,E1 -8154.553,E2 -8154.553} C_VEL
LIN {X 0,Y 460.511,Z 141.117,A -85,B 0,C 180,E1 -8157.714,E2 -8157.714} C_VEL
LIN {X 0,Y 460.509,Z 141.126,A -85,B 0,C 180,E1 -8160.767,E2 -8160.767} C_VEL
LIN {X 0,Y 460.528,Z 141.117,A -85,B 0,C 180,E1 -8164.206,E2 -8164.206} C_VEL
LIN {X 0,Y 460.496,Z 141.119,A -85,B 0,C 180,E1 -8167.57,E2 -8167.57} C_VEL
LIN {X 0,Y 460.554,Z 141.118,A -85,B 0,C 180,E1 -8170.384,E2 -8170.384} C_VEL
LIN {X 0,Y 460.559,Z 141.114,A -85,B 0,C 180,E1 -8174.057,E2 -8174.057} C_VEL
LIN {X 0,Y 460.595,Z 141.108,A -85,B 0,C 180,E1 -8177.665,E2 -8177.665} C_VEL
LIN {X 0,Y 460.542,Z 141.113,A -85,B 0,C 180,E1 -8179.185,E2 -8179.185} C_VEL
LIN {X 0,Y 459.876,Z 141.201,A -85,B 0,C 180,E1 -8179.915,E2 -8179.915} C_VEL
LIN {X 0,Y 457.045,Z 141.55,A -85,B 0,C 180,E1 -8181.101,E2 -8181.101} C_VEL
LIN {X 0,Y 454.662,Z 141.851,A -85,B 0,C 180,E1 -8182.058,E2 -8182.058} C_VEL
LIN {X 0,Y 453.651,Z 141.974,A -85,B 0,C 180,E1 -8182.797,E2 -8182.797} C_VEL
LIN {X 0,Y 453.575,Z 141.982,A -85,B 0,C 180,E1 -8183.047,E2 -8183.047} C_VEL
LIN {X 0,Y 453.638,Z 141.976,A -85,B 0,C 180,E1 -8184.666,E2 -8184.666} C_VEL
LIN {X 0,Y 453.679,Z 141.977,A -85,B 0,C 180,E1 -8188.224,E2 -8188.224} C_VEL
LIN {X 0,Y 453.629,Z 141.982,A -85,B 0,C 180,E1 -8190.444,E2 -8190.444} C_VEL
LIN {X 0,Y 453.587,Z 141.998,A -85,B 0,C 180,E1 -8190.666,E2 -8190.666} C_VEL
LIN {X 0,Y 454.747,Z 148.915,A -85,B 0,C 180,E1 -8192.214,E2 -8192.214} C_VEL
LIN {X 0,Y 454.541,Z 159.776,A -85,B 0,C 180,E1 -8194.517,E2 -8194.517} C_VEL
LIN {X 0,Y 457.742,Z 175.968,A -85,B 0,C 180,E1 -8194.927,E2 -8194.927} C_VEL
LIN {X 0,Y 456.871,Z 267.443,A -85,B 0,C 180,E1 -8196.403,E2 -8196.403} C_VEL
LIN {X 0,Y 456.51,Z 280.629,A -85,B 0,C 180,E1 -8196.797,E2 -8196.797} C_VEL
LIN {X 0,Y 456.206,Z 293.177,A -85,B 0,C 180,E1 -8197.357,E2 -8197.357} C_VEL
LIN {X 0,Y 455.737,Z 305.056,A -85,B 0,C 180,E1 -8198.077,E2 -8198.077} C_VEL
LIN {X 0,Y 455.215,Z 316.622,A -85,B 0,C 180,E1 -8198.982,E2 -8198.982} C_VEL
LIN {X 0,Y 454.676,Z 327.148,A -85,B 0,C 180,E1 -8200.014,E2 -8200.014} C_VEL
LIN {X 0,Y 454.082,Z 336.502,A -85,B 0,C 180,E1 -8201.155,E2 -8201.155} C_VEL
LIN {X 0,Y 453.574,Z 345.635,A -85,B 0,C 180,E1 -8202.539,E2 -8202.539} C_VEL
LIN {X 0,Y 453.205,Z 352.839,A -85,B 0,C 180,E1 -8203.908,E2 -8203.908} C_VEL
LIN {X 0,Y 452.891,Z 358.622,A -85,B 0,C 180,E1 -8205.296,E2 -8205.296} C_VEL
LIN {X 0,Y 452.697,Z 363.15,A -85,B 0,C 180,E1 -8206.691,E2 -8206.691} C_VEL
LIN {X 0,Y 452.529,Z 366.552,A -85,B 0,C 180,E1 -8208.096,E2 -8208.096} C_VEL
LIN {X 0,Y 452.47,Z 368.233,A -85,B 0,C 180,E1 -8209.037,E2 -8209.037} C_VEL
LIN {X 0,Y 452.39,Z 369.462,A -85,B 0,C 180,E1 -8209.985,E2 -8209.985} C_VEL
LIN {X 0,Y 452.351,Z 370.363,A -85,B 0,C 180,E1 -8211.223,E2 -8211.223} C_VEL
LIN {X 0,Y 452.35,Z 370.395,A -85,B 0,C 180,E1 -8212.856,E2 -8212.856} C_VEL
LIN {X 0,Y 452.395,Z 369.765,A -85,B 0,C 180,E1 -8213.823,E2 -8213.823} C_VEL
LIN {X 0,Y 452.432,Z 368.69,A -85,B 0,C 180,E1 -8214.798,E2 -8214.798} C_VEL
LIN {X 0,Y 452.613,Z 366.124,A -85,B 0,C 180,E1 -8216.266,E2 -8216.266} C_VEL
LIN {X 0,Y 452.805,Z 362.197,A -85,B 0,C 180,E1 -8217.788,E2 -8217.788} C_VEL
LIN {X 0,Y 452.982,Z 357.171,A -85,B 0,C 180,E1 -8219.231,E2 -8219.231} C_VEL
LIN {X 0,Y 453.351,Z 350.244,A -85,B 0,C 180,E1 -8220.769,E2 -8220.769} C_VEL
LIN {X 0,Y 453.765,Z 343.053,A -85,B 0,C 180,E1 -8222.037,E2 -8222.037} C_VEL
LIN {X 0,Y 454.298,Z 333.8,A -85,B 0,C 180,E1 -8223.346,E2 -8223.346} C_VEL
LIN {X 0,Y 454.827,Z 324.008,A -85,B 0,C 180,E1 -8224.467,E2 -8224.467} C_VEL
LIN {X 0,Y 455.428,Z 313.545,A -85,B 0,C 180,E1 -8225.431,E2 -8225.431} C_VEL
LIN {X 0,Y 455.942,Z 302.108,A -85,B 0,C 180,E1 -8226.265,E2 -8226.265} C_VEL
LIN {X 0,Y 456.475,Z 289.441,A -85,B 0,C 180,E1 -8226.971,E2 -8226.971} C_VEL
LIN {X 0,Y 456.805,Z 276.879,A -85,B 0,C 180,E1 -8227.476,E2 -8227.476} C_VEL
LIN {X 0,Y 457.036,Z 264.28,A -85,B 0,C 180,E1 -8227.802,E2 -8227.802} C_VEL
LIN {X 0,Y 457.862,Z 175.564,A -85,B 0,C 180,E1 -8229.225,E2 -8229.225} C_VEL
LIN {X 0,Y 454.705,Z 160.077,A -85,B 0,C 180,E1 -8229.615,E2 -8229.615} C_VEL
LIN {X 0,Y 454.931,Z 150.379,A -85,B 0,C 180,E1 -8231.628,E2 -8231.628} C_VEL
LIN {X 0,Y 453.534,Z 141.994,A -85,B 0,C 180,E1 -8233.486,E2 -8233.486} C_VEL
LIN {X 0,Y 453.488,Z 141.993,A -85,B 0,C 180,E1 -8237.009,E2 -8237.009} C_VEL
LIN {X 0,Y 453.525,Z 141.99,A -85,B 0,C 180,E1 -8240.555,E2 -8240.555} C_VEL
LIN {X 0,Y 453.451,Z 142.004,A -85,B 0,C 180,E1 -8243.918,E2 -8243.918} C_VEL
LIN {X 0,Y 453.48,Z 141.998,A -85,B 0,C 180,E1 -8247.152,E2 -8247.152} C_VEL
LIN {X 0,Y 453.473,Z 141.994,A -85,B 0,C 180,E1 -8250.269,E2 -8250.269} C_VEL
LIN {X 0,Y 453.506,Z 141.996,A -85,B 0,C 180,E1 -8253.295,E2 -8253.295} C_VEL
LIN {X 0,Y 453.502,Z 141.991,A -85,B 0,C 180,E1 -8256.24,E2 -8256.24} C_VEL
LIN {X 0,Y 453.482,Z 141.998,A -85,B 0,C 180,E1 -8259.119,E2 -8259.119} C_VEL
LIN {X 0,Y 453.501,Z 141.991,A -85,B 0,C 180,E1 -8261.945,E2 -8261.945} C_VEL
LIN {X 0,Y 453.539,Z 141.991,A -85,B 0,C 180,E1 -8264.727,E2 -8264.727} C_VEL
LIN {X 0,Y 453.56,Z 141.986,A -85,B 0,C 180,E1 -8268.38,E2 -8268.38} C_VEL
LIN {X 0,Y 453.586,Z 141.98,A -85,B 0,C 180,E1 -8271.087,E2 -8271.087} C_VEL
LIN {X 0,Y 453.654,Z 141.972,A -85,B 0,C 180,E1 -8273.775,E2 -8273.775} C_VEL
LIN {X 0,Y 453.737,Z 141.96,A -85,B 0,C 180,E1 -8277.337,E2 -8277.337} C_VEL
LIN {X 0,Y 453.82,Z 141.951,A -85,B 0,C 180,E1 -8280.001,E2 -8280.001} C_VEL
LIN {X 0,Y 453.708,Z 141.967,A -85,B 0,C 180,E1 -8282.664,E2 -8282.664} C_VEL
LIN {X 0,Y 453.644,Z 141.972,A -85,B 0,C 180,E1 -8286.226,E2 -8286.226} C_VEL
LIN {X 0,Y 453.58,Z 141.98,A -85,B 0,C 180,E1 -8288.914,E2 -8288.914} C_VEL
LIN {X 0,Y 453.567,Z 141.984,A -85,B 0,C 180,E1 -8292.529,E2 -8292.529} C_VEL
LIN {X 0,Y 453.505,Z 141.99,A -85,B 0,C 180,E1 -8296.091,E2 -8296.091} C_VEL
LIN {X 0,Y 453.52,Z 141.99,A -85,B 0,C 180,E1 -8299.04,E2 -8299.04} C_VEL
LIN {X 0,Y 453.473,Z 141.996,A -85,B 0,C 180,E1 -8301.837,E2 -8301.837} C_VEL
LIN {X 0,Y 453.471,Z 141.995,A -85,B 0,C 180,E1 -8304.738,E2 -8304.738} C_VEL
LIN {X 0,Y 453.459,Z 141.999,A -85,B 0,C 180,E1 -8307.942,E2 -8307.942} C_VEL
LIN {X 0,Y 453.449,Z 141.995,A -85,B 0,C 180,E1 -8310.762,E2 -8310.762} C_VEL
LIN {X 0,Y 453.455,Z 141.995,A -85,B 0,C 180,E1 -8313.915,E2 -8313.915} C_VEL
LIN {X 0,Y 453.433,Z 142.004,A -85,B 0,C 180,E1 -8317.192,E2 -8317.192} C_VEL
LIN {X 0,Y 453.466,Z 142,A -85,B 0,C 180,E1 -8320.613,E2 -8320.613} C_VEL
LIN {X 0,Y 453.483,Z 141.997,A -85,B 0,C 180,E1 -8324.529,E2 -8324.529} C_VEL
LIN {X 0,Y 453.437,Z 142.004,A -85,B 0,C 180,E1 -8328.071,E2 -8328.071} C_VEL
LIN {X 0,Y 453.443,Z 142.005,A -85,B 0,C 180,E1 -8330.802,E2 -8330.802} C_VEL
LIN {X 0,Y 453.451,Z 141.996,A -85,B 0,C 180,E1 -8333.917,E2 -8333.917} C_VEL
LIN {X 0,Y 453.477,Z 141.998,A -85,B 0,C 180,E1 -8337.151,E2 -8337.151} C_VEL
LIN {X 0,Y 453.465,Z 142.001,A -85,B 0,C 180,E1 -8340.268,E2 -8340.268} C_VEL
LIN {X 0,Y 453.504,Z 142.107,A -85,B 0,C 180,E1 -8343.576,E2 -8343.576} C_VEL
LIN {X 0,Y 455.841,Z 154.144,A -85,B 0,C 180,E1 -8345.934,E2 -8345.934} C_VEL
LIN {X 0,Y 455.605,Z 161.777,A -85,B 0,C 180,E1 -8347.317,E2 -8347.317} C_VEL
LIN {X 0,Y 454.833,Z 178.963,A -85,B 0,C 180,E1 -8350.381,E2 -8350.381} C_VEL
LIN {X 0,Y 454.351,Z 190.404,A -85,B 0,C 180,E1 -8352.398,E2 -8352.398} C_VEL
LIN {X 0,Y 457.606,Z 213.059,A -85,B 0,C 180,E1 -8352.907,E2 -8352.907} C_VEL
LIN {X 0,Y 456.868,Z 299.059,A -85,B 0,C 180,E1 -8354.297,E2 -8354.297} C_VEL
LIN {X 0,Y 456.467,Z 312.275,A -85,B 0,C 180,E1 -8354.684,E2 -8354.684} C_VEL
LIN {X 0,Y 455.934,Z 324.425,A -85,B 0,C 180,E1 -8355.209,E2 -8355.209} C_VEL
LIN {X 0,Y 455.359,Z 336.704,A -85,B 0,C 180,E1 -8355.931,E2 -8355.931} C_VEL
LIN {X 0,Y 454.802,Z 347.923,A -85,B 0,C 180,E1 -8356.79,E2 -8356.79} C_VEL
LIN {X 0,Y 454.249,Z 358.787,A -85,B 0,C 180,E1 -8357.831,E2 -8357.831} C_VEL
LIN {X 0,Y 453.773,Z 367.35,A -85,B 0,C 180,E1 -8358.837,E2 -8358.837} C_VEL
LIN {X 0,Y 453.305,Z 375.254,A -85,B 0,C 180,E1 -8359.955,E2 -8359.955} C_VEL
LIN {X 0,Y 452.982,Z 382.981,A -85,B 0,C 180,E1 -8361.3,E2 -8361.3} C_VEL
LIN {X 0,Y 452.675,Z 390.109,A -85,B 0,C 180,E1 -8362.865,E2 -8362.865} C_VEL
LIN {X 0,Y 452.532,Z 394.853,A -85,B 0,C 180,E1 -8364.206,E2 -8364.206} C_VEL
LIN {X 0,Y 452.485,Z 398.481,A -85,B 0,C 180,E1 -8365.546,E2 -8365.546} C_VEL
LIN {X 0,Y 452.482,Z 400.352,A -85,B 0,C 180,E1 -8366.438,E2 -8366.438} C_VEL
LIN {X 0,Y 452.509,Z 401.757,A -85,B 0,C 180,E1 -8367.33,E2 -8367.33} C_VEL
LIN {X 0,Y 452.461,Z 403.372,A -85,B 0,C 180,E1 -8369.11,E2 -8369.11} C_VEL
LIN {X 0,Y 452.47,Z 403.589,A -85,B 0,C 180,E1 -8370,E2 -8370} C_VEL
LIN {X 0,Y 452.46,Z 403.37,A -85,B 0,C 180,E1 -8370.89,E2 -8370.89} C_VEL
LIN {X 0,Y 452.509,Z 401.761,A -85,B 0,C 180,E1 -8372.671,E2 -8372.671} C_VEL
LIN {X 0,Y 452.482,Z 400.352,A -85,B 0,C 180,E1 -8373.562,E2 -8373.562} C_VEL
LIN {X 0,Y 452.542,Z 397.399,A -85,B 0,C 180,E1 -8374.9,E2 -8374.9} C_VEL
LIN {X 0,Y 452.612,Z 392.849,A -85,B 0,C 180,E1 -8376.396,E2 -8376.396} C_VEL
LIN {X 0,Y 452.798,Z 387.236,A -85,B 0,C 180,E1 -8377.806,E2 -8377.806} C_VEL
LIN {X 0,Y 453.052,Z 380.511,A -85,B 0,C 180,E1 -8379.149,E2 -8379.149} C_VEL
LIN {X 0,Y 453.431,Z 372.168,A -85,B 0,C 180,E1 -8380.494,E2 -8380.494} C_VEL
LIN {X 0,Y 453.947,Z 363.595,A -85,B 0,C 180,E1 -8381.611,E2 -8381.611} C_VEL
LIN {X 0,Y 454.535,Z 352.651,A -85,B 0,C 180,E1 -8382.764,E2 -8382.764} C_VEL
LIN {X 0,Y 454.992,Z 342.527,A -85,B 0,C 180,E1 -8383.625,E2 -8383.625} C_VEL
LIN {X 0,Y 455.597,Z 330.995,A -85,B 0,C 180,E1 -8384.403,E2 -8384.403} C_VEL
LIN {X 0,Y 456.133,Z 319.036,A -85,B 0,C 180,E1 -8385.014,E2 -8385.014} C_VEL
LIN {X 0,Y 456.597,Z 306.125,A -85,B 0,C 180,E1 -8385.484,E2 -8385.484} C_VEL
LIN {X 0,Y 456.893,Z 292.485,A -85,B 0,C 180,E1 -8385.788,E2 -8385.788} C_VEL
LIN {X 0,Y 457.444,Z 211.138,A -85,B 0,C 180,E1 -8387.084,E2 -8387.084} C_VEL
LIN {X 0,Y 454.35,Z 190.849,A -85,B 0,C 180,E1 -8387.533,E2 -8387.533} C_VEL
LIN {X 0,Y 455.058,Z 173.749,A -85,B 0,C 180,E1 -8390.571,E2 -8390.571} C_VEL
LIN {X 0,Y 455.783,Z 159.373,A -85,B 0,C 180,E1 -8393.154,E2 -8393.154} C_VEL
LIN {X 0,Y 455.901,Z 154.33,A -85,B 0,C 180,E1 -8394.075,E2 -8394.075} C_VEL
LIN {X 0,Y 453.491,Z 141.998,A -85,B 0,C 180,E1 -8396.525,E2 -8396.525} C_VEL
LIN {X 0,Y 453.473,Z 142.002,A -85,B 0,C 180,E1 -8399.784,E2 -8399.784} C_VEL
LIN {X 0,Y 453.485,Z 141.995,A -85,B 0,C 180,E1 -8403.187,E2 -8403.187} C_VEL
LIN {X 0,Y 453.454,Z 141.997,A -85,B 0,C 180,E1 -8406.298,E2 -8406.298} C_VEL
LIN {X 0,Y 453.453,Z 142.004,A -85,B 0,C 180,E1 -8409.454,E2 -8409.454} C_VEL
LIN {X 0,Y 453.44,Z 142,A -85,B 0,C 180,E1 -8411.929,E2 -8411.929} C_VEL
LIN {X 0,Y 453.486,Z 141.998,A -85,B 0,C 180,E1 -8415.472,E2 -8415.472} C_VEL
LIN {X 0,Y 453.475,Z 141.999,A -85,B 0,C 180,E1 -8419.388,E2 -8419.388} C_VEL
LIN {X 0,Y 453.454,Z 142,A -85,B 0,C 180,E1 -8422.81,E2 -8422.81} C_VEL
LIN {X 0,Y 453.472,Z 141.994,A -85,B 0,C 180,E1 -8426.086,E2 -8426.086} C_VEL
LIN {X 0,Y 453.459,Z 142,A -85,B 0,C 180,E1 -8429.239,E2 -8429.239} C_VEL
LIN {X 0,Y 453.494,Z 141.993,A -85,B 0,C 180,E1 -8432.294,E2 -8432.294} C_VEL
LIN {X 0,Y 453.474,Z 141.996,A -85,B 0,C 180,E1 -8435.263,E2 -8435.263} C_VEL
LIN {X 0,Y 453.484,Z 141.996,A -85,B 0,C 180,E1 -8438.416,E2 -8438.416} C_VEL
LIN {X 0,Y 453.528,Z 141.991,A -85,B 0,C 180,E1 -8441.008,E2 -8441.008} C_VEL
LIN {X 0,Y 453.523,Z 141.994,A -85,B 0,C 180,E1 -8444.725,E2 -8444.725} C_VEL
LIN {X 0,Y 453.563,Z 141.989,A -85,B 0,C 180,E1 -8448.378,E2 -8448.378} C_VEL
LIN {X 0,Y 453.57,Z 141.983,A -85,B 0,C 180,E1 -8451.086,E2 -8451.086} C_VEL
LIN {X 0,Y 453.64,Z 141.975,A -85,B 0,C 180,E1 -8453.773,E2 -8453.773} C_VEL
LIN {X 0,Y 453.707,Z 141.965,A -85,B 0,C 180,E1 -8457.336,E2 -8457.336} C_VEL
LIN {X 0,Y 453.793,Z 141.959,A -85,B 0,C 180,E1 -8459.999,E2 -8459.999} C_VEL
LIN {X 0,Y 453.706,Z 141.967,A -85,B 0,C 180,E1 -8462.663,E2 -8462.663} C_VEL
LIN {X 0,Y 453.638,Z 141.979,A -85,B 0,C 180,E1 -8466.225,E2 -8466.225} C_VEL
LIN {X 0,Y 453.561,Z 141.983,A -85,B 0,C 180,E1 -8468.913,E2 -8468.913} C_VEL
LIN {X 0,Y 453.567,Z 141.984,A -85,B 0,C 180,E1 -8472.528,E2 -8472.528} C_VEL
LIN {X 0,Y 453.498,Z 141.994,A -85,B 0,C 180,E1 -8476.197,E2 -8476.197} C_VEL
LIN {X 0,Y 453.487,Z 141.993,A -85,B 0,C 180,E1 -8479.026,E2 -8479.026} C_VEL
LIN {X 0,Y 453.472,Z 142,A -85,B 0,C 180,E1 -8481.835,E2 -8481.835} C_VEL
LIN {X 0,Y 453.469,Z 141.995,A -85,B 0,C 180,E1 -8484.736,E2 -8484.736} C_VEL
LIN {X 0,Y 453.46,Z 141.999,A -85,B 0,C 180,E1 -8487.941,E2 -8487.941} C_VEL
LIN {X 0,Y 453.453,Z 141.997,A -85,B 0,C 180,E1 -8490.76,E2 -8490.76} C_VEL
LIN {X 0,Y 453.465,Z 141.997,A -85,B 0,C 180,E1 -8493.913,E2 -8493.913} C_VEL
LIN {X 0,Y 453.444,Z 142.004,A -85,B 0,C 180,E1 -8497.189,E2 -8497.189} C_VEL
LIN {X 0,Y 453.467,Z 141.996,A -85,B 0,C 180,E1 -8500.611,E2 -8500.611} C_VEL
LIN {X 0,Y 453.478,Z 141.995,A -85,B 0,C 180,E1 -8504.527,E2 -8504.527} C_VEL
LIN {X 0,Y 453.431,Z 141.999,A -85,B 0,C 180,E1 -8508.07,E2 -8508.07} C_VEL
LIN {X 0,Y 453.46,Z 142.001,A -85,B 0,C 180,E1 -8510.797,E2 -8510.797} C_VEL
LIN {X 0,Y 453.445,Z 141.998,A -85,B 0,C 180,E1 -8513.916,E2 -8513.916} C_VEL
LIN {X 0,Y 453.468,Z 141.999,A -85,B 0,C 180,E1 -8517.15,E2 -8517.15} C_VEL
LIN {X 0,Y 453.45,Z 141.999,A -85,B 0,C 180,E1 -8520.266,E2 -8520.266} C_VEL
LIN {X 0,Y 453.435,Z 142,A -85,B 0,C 180,E1 -8523.289,E2 -8523.289} C_VEL
LIN {X 0,Y 453.485,Z 141.996,A -85,B 0,C 180,E1 -8526.237,E2 -8526.237} C_VEL
LIN {X 0,Y 453.467,Z 141.996,A -85,B 0,C 180,E1 -8529.117,E2 -8529.117} C_VEL
LIN {X 0,Y 453.475,Z 141.995,A -85,B 0,C 180,E1 -8531.943,E2 -8531.943} C_VEL
LIN {X 0,Y 453.511,Z 141.993,A -85,B 0,C 180,E1 -8534.725,E2 -8534.725} C_VEL
LIN {X 0,Y 453.536,Z 141.994,A -85,B 0,C 180,E1 -8538.378,E2 -8538.378} C_VEL
LIN {X 0,Y 453.55,Z 141.985,A -85,B 0,C 180,E1 -8541.086,E2 -8541.086} C_VEL
LIN {X 0,Y 453.575,Z 141.982,A -85,B 0,C 180,E1 -8543.047,E2 -8543.047} C_VEL
LIN {X 0,Y 452.893,Z 142.071,A -85,B 0,C 180,E1 -8543.788,E2 -8543.788} C_VEL
LIN {X 0,Y 449.944,Z 142.435,A -85,B 0,C 180,E1 -8544.99,E2 -8544.99} C_VEL
LIN {X 0,Y 447.515,Z 142.741,A -85,B 0,C 180,E1 -8545.96,E2 -8545.96} C_VEL
LIN {X 0,Y 446.571,Z 142.859,A -85,B 0,C 180,E1 -8546.71,E2 -8546.71} C_VEL
LIN {X 0,Y 446.549,Z 142.86,A -85,B 0,C 180,E1 -8546.964,E2 -8546.964} C_VEL
LIN {X 0,Y 446.708,Z 142.845,A -85,B 0,C 180,E1 -8550,E2 -8550} C_VEL
LIN {X 0,Y 446.606,Z 143.006,A -85,B 0,C 180,E1 -8550.507,E2 -8550.507} C_VEL
LIN {X 0,Y 447.817,Z 150.687,A -85,B 0,C 180,E1 -8552.248,E2 -8552.248} C_VEL
LIN {X 0,Y 447.582,Z 160.051,A -85,B 0,C 180,E1 -8554.249,E2 -8554.249} C_VEL
LIN {X 0,Y 450.9,Z 176.209,A -85,B 0,C 180,E1 -8554.666,E2 -8554.666} C_VEL
LIN {X 0,Y 450.038,Z 267.537,A -85,B 0,C 180,E1 -8556.163,E2 -8556.163} C_VEL
LIN {X 0,Y 449.661,Z 280.776,A -85,B 0,C 180,E1 -8556.563,E2 -8556.563} C_VEL
LIN {X 0,Y 449.329,Z 293.363,A -85,B 0,C 180,E1 -8557.132,E2 -8557.132} C_VEL
LIN {X 0,Y 448.851,Z 305.421,A -85,B 0,C 180,E1 -8557.874,E2 -8557.874} C_VEL
LIN {X 0,Y 448.297,Z 316.559,A -85,B 0,C 180,E1 -8558.756,E2 -8558.756} C_VEL
LIN {X 0,Y 447.732,Z 327.368,A -85,B 0,C 180,E1 -8559.829,E2 -8559.829} C_VEL
LIN {X 0,Y 447.175,Z 335.894,A -85,B 0,C 180,E1 -8560.871,E2 -8560.871} C_VEL
LIN {X 0,Y 446.601,Z 344.711,A -85,B 0,C 180,E1 -8562.196,E2 -8562.196} C_VEL
LIN {X 0,Y 446.186,Z 352.541,A -85,B 0,C 180,E1 -8563.666,E2 -8563.666} C_VEL
LIN {X 0,Y 445.863,Z 358.451,A -85,B 0,C 180,E1 -8565.075,E2 -8565.075} C_VEL
LIN {X 0,Y 445.645,Z 363.077,A -85,B 0,C 180,E1 -8566.491,E2 -8566.491} C_VEL
LIN {X 0,Y 445.525,Z 365.518,A -85,B 0,C 180,E1 -8567.441,E2 -8567.441} C_VEL
LIN {X 0,Y 445.403,Z 368.158,A -85,B 0,C 180,E1 -8568.787,E2 -8568.787} C_VEL
LIN {X 0,Y 445.277,Z 370.04,A -85,B 0,C 180,E1 -8570.318,E2 -8570.318} C_VEL
LIN {X 0,Y 445.26,Z 370.69,A -85,B 0,C 180,E1 -8571.371,E2 -8571.371} C_VEL
LIN {X 0,Y 445.266,Z 370.786,A -85,B 0,C 180,E1 -8572.26,E2 -8572.26} C_VEL
LIN {X 0,Y 445.306,Z 370.124,A -85,B 0,C 180,E1 -8573.743,E2 -8573.743} C_VEL
LIN {X 0,Y 445.39,Z 368.406,A -85,B 0,C 180,E1 -8575.217,E2 -8575.217} C_VEL
LIN {X 0,Y 445.575,Z 365.532,A -85,B 0,C 180,E1 -8576.713,E2 -8576.713} C_VEL
LIN {X 0,Y 445.785,Z 361.393,A -85,B 0,C 180,E1 -8578.227,E2 -8578.227} C_VEL
LIN {X 0,Y 446.009,Z 356.453,A -85,B 0,C 180,E1 -8579.598,E2 -8579.598} C_VEL
LIN {X 0,Y 446.362,Z 349.869,A -85,B 0,C 180,E1 -8581.041,E2 -8581.041} C_VEL
LIN {X 0,Y 446.83,Z 342.493,A -85,B 0,C 180,E1 -8582.328,E2 -8582.328} C_VEL
LIN {X 0,Y 447.381,Z 333.229,A -85,B 0,C 180,E1 -8583.636,E2 -8583.636} C_VEL
LIN {X 0,Y 447.989,Z 323.045,A -85,B 0,C 180,E1 -8584.795,E2 -8584.795} C_VEL
LIN {X 0,Y 448.662,Z 311.443,A -85,B 0,C 180,E1 -8585.835,E2 -8585.835} C_VEL
LIN {X 0,Y 449.178,Z 300.805,A -85,B 0,C 180,E1 -8586.592,E2 -8586.592} C_VEL
LIN {X 0,Y 449.656,Z 289.736,A -85,B 0,C 180,E1 -8587.207,E2 -8587.207} C_VEL
LIN {X 0,Y 450,Z 277.243,A -85,B 0,C 180,E1 -8587.718,E2 -8587.718} C_VEL
LIN {X 0,Y 450.243,Z 264.718,A -85,B 0,C 180,E1 -8588.048,E2 -8588.048} C_VEL
LIN {X 0,Y 451.054,Z 176.184,A -85,B 0,C 180,E1 -8589.494,E2 -8589.494} C_VEL
LIN {X 0,Y 447.782,Z 160.295,A -85,B 0,C 180,E1 -8589.91,E2 -8589.91} C_VEL
LIN {X 0,Y 447.993,Z 151.248,A -85,B 0,C 180,E1 -8591.815,E2 -8591.815} C_VEL
LIN {X 0,Y 446.468,Z 142.875,A -85,B 0,C 180,E1 -8593.723,E2 -8593.723} C_VEL
LIN {X 0,Y 446.443,Z 142.873,A -85,B 0,C 180,E1 -8596.398,E2 -8596.398} C_VEL
LIN {X 0,Y 446.464,Z 142.878,A -85,B 0,C 180,E1 -8599.806,E2 -8599.806} C_VEL
LIN {X 0,Y 446.428,Z 142.88,A -85,B 0,C 180,E1 -8602.124,E2 -8602.124} C_VEL
LIN {X 0,Y 446.427,Z 142.881,A -85,B 0,C 180,E1 -8605.478,E2 -8605.478} C_VEL
LIN {X 0,Y 446.414,Z 142.875,A -85,B 0,C 180,E1 -8608.701,E2 -8608.701} C_VEL
LIN {X 0,Y 446.483,Z 142.869,A -85,B 0,C 180,E1 -8611.822,E2 -8611.822} C_VEL
LIN {X 0,Y 446.457,Z 142.874,A -85,B 0,C 180,E1 -8614.849,E2 -8614.849} C_VEL
LIN {X 0,Y 446.448,Z 142.871,A -85,B 0,C 180,E1 -8618.246,E2 -8618.246} C_VEL
LIN {X 0,Y 446.45,Z 142.87,A -85,B 0,C 180,E1 -8621.65,E2 -8621.65} C_VEL
LIN {X 0,Y 446.507,Z 142.865,A -85,B 0,C 180,E1 -8624.481,E2 -8624.481} C_VEL
LIN {X 0,Y 446.518,Z 142.861,A -85,B 0,C 180,E1 -8628.194,E2 -8628.194} C_VEL
LIN {X 0,Y 446.533,Z 142.859,A -85,B 0,C 180,E1 -8630.945,E2 -8630.945} C_VEL
LIN {X 0,Y 446.622,Z 142.848,A -85,B 0,C 180,E1 -8633.677,E2 -8633.677} C_VEL
LIN {X 0,Y 446.684,Z 142.839,A -85,B 0,C 180,E1 -8637.295,E2 -8637.295} C_VEL
LIN {X 0,Y 446.789,Z 142.827,A -85,B 0,C 180,E1 -8640.001,E2 -8640.001} C_VEL
LIN {X 0,Y 446.658,Z 142.845,A -85,B 0,C 180,E1 -8642.706,E2 -8642.706} C_VEL
LIN {X 0,Y 446.613,Z 142.848,A -85,B 0,C 180,E1 -8646.325,E2 -8646.325} C_VEL
LIN {X 0,Y 446.529,Z 142.858,A -85,B 0,C 180,E1 -8649.056,E2 -8649.056} C_VEL
LIN {X 0,Y 446.524,Z 142.86,A -85,B 0,C 180,E1 -8652.73,E2 -8652.73} C_VEL
LIN {X 0,Y 446.456,Z 142.867,A -85,B 0,C 180,E1 -8656.209,E2 -8656.209} C_VEL
LIN {X 0,Y 446.469,Z 142.87,A -85,B 0,C 180,E1 -8659.304,E2 -8659.304} C_VEL
LIN {X 0,Y 446.41,Z 142.875,A -85,B 0,C 180,E1 -8662.201,E2 -8662.201} C_VEL
LIN {X 0,Y 446.423,Z 142.875,A -85,B 0,C 180,E1 -8665.155,E2 -8665.155} C_VEL
LIN {X 0,Y 446.417,Z 142.875,A -85,B 0,C 180,E1 -8668.184,E2 -8668.184} C_VEL
LIN {X 0,Y 446.39,Z 142.879,A -85,B 0,C 180,E1 -8671.303,E2 -8671.303} C_VEL
LIN {X 0,Y 446.413,Z 142.872,A -85,B 0,C 180,E1 -8674.525,E2 -8674.525} C_VEL
LIN {X 0,Y 446.388,Z 142.876,A -85,B 0,C 180,E1 -8677.882,E2 -8677.882} C_VEL
LIN {X 0,Y 446.397,Z 142.882,A -85,B 0,C 180,E1 -8681.395,E2 -8681.395} C_VEL
LIN {X 0,Y 446.451,Z 142.879,A -85,B 0,C 180,E1 -8685.104,E2 -8685.104} C_VEL
LIN {X 0,Y 446.402,Z 142.884,A -85,B 0,C 180,E1 -8688.606,E2 -8688.606} C_VEL
LIN {X 0,Y 446.406,Z 142.877,A -85,B 0,C 180,E1 -8691.923,E2 -8691.923} C_VEL
LIN {X 0,Y 446.424,Z 142.874,A -85,B 0,C 180,E1 -8695.477,E2 -8695.477} C_VEL
LIN {X 0,Y 446.417,Z 142.878,A -85,B 0,C 180,E1 -8698.7,E2 -8698.7} C_VEL
LIN {X 0,Y 446.427,Z 142.877,A -85,B 0,C 180,E1 -8701.836,E2 -8701.836} C_VEL
LIN {X 0,Y 446.441,Z 142.989,A -85,B 0,C 180,E1 -8703.336,E2 -8703.336} C_VEL
LIN {X 0,Y 448.773,Z 154.666,A -85,B 0,C 180,E1 -8705.671,E2 -8705.671} C_VEL
LIN {X 0,Y 448.915,Z 158.926,A -85,B 0,C 180,E1 -8706.471,E2 -8706.471} C_VEL
LIN {X 0,Y 448.06,Z 174.693,A -85,B 0,C 180,E1 -8709.334,E2 -8709.334} C_VEL
LIN {X 0,Y 447.367,Z 190.162,A -85,B 0,C 180,E1 -8712.113,E2 -8712.113} C_VEL
LIN {X 0,Y 450.842,Z 213.253,A -85,B 0,C 180,E1 -8712.643,E2 -8712.643} C_VEL
LIN {X 0,Y 450.042,Z 299.002,A -85,B 0,C 180,E1 -8714.053,E2 -8714.053} C_VEL
LIN {X 0,Y 449.619,Z 312.143,A -85,B 0,C 180,E1 -8714.445,E2 -8714.445} C_VEL
LIN {X 0,Y 449.029,Z 325.37,A -85,B 0,C 180,E1 -8715.034,E2 -8715.034} C_VEL
LIN {X 0,Y 448.459,Z 336.5,A -85,B 0,C 180,E1 -8715.71,E2 -8715.71} C_VEL
LIN {X 0,Y 447.875,Z 347.139,A -85,B 0,C 180,E1 -8716.531,E2 -8716.531} C_VEL
LIN {X 0,Y 447.271,Z 358.564,A -85,B 0,C 180,E1 -8717.638,E2 -8717.638} C_VEL
LIN {X 0,Y 446.785,Z 367.121,A -85,B 0,C 180,E1 -8718.66,E2 -8718.66} C_VEL
LIN {X 0,Y 446.263,Z 375.018,A -85,B 0,C 180,E1 -8719.795,E2 -8719.795} C_VEL
LIN {X 0,Y 445.933,Z 382.738,A -85,B 0,C 180,E1 -8721.161,E2 -8721.161} C_VEL
LIN {X 0,Y 445.603,Z 389.862,A -85,B 0,C 180,E1 -8722.752,E2 -8722.752} C_VEL
LIN {X 0,Y 445.446,Z 394.197,A -85,B 0,C 180,E1 -8723.986,E2 -8723.986} C_VEL
LIN {X 0,Y 445.411,Z 398.229,A -85,B 0,C 180,E1 -8725.475,E2 -8725.475} C_VEL
LIN {X 0,Y 445.381,Z 400.098,A -85,B 0,C 180,E1 -8726.381,E2 -8726.381} C_VEL
LIN {X 0,Y 445.433,Z 401.502,A -85,B 0,C 180,E1 -8727.287,E2 -8727.287} C_VEL
LIN {X 0,Y 445.369,Z 403.115,A -85,B 0,C 180,E1 -8729.096,E2 -8729.096} C_VEL
LIN {X 0,Y 445.376,Z 403.33,A -85,B 0,C 180,E1 -8730,E2 -8730} C_VEL
LIN {X 0,Y 445.369,Z 403.108,A -85,B 0,C 180,E1 -8730.904,E2 -8730.904} C_VEL
LIN {X 0,Y 445.434,Z 401.497,A -85,B 0,C 180,E1 -8732.713,E2 -8732.713} C_VEL
LIN {X 0,Y 445.381,Z 400.084,A -85,B 0,C 180,E1 -8733.619,E2 -8733.619} C_VEL
LIN {X 0,Y 445.47,Z 397.128,A -85,B 0,C 180,E1 -8734.978,E2 -8734.978} C_VEL
LIN {X 0,Y 445.492,Z 393.12,A -85,B 0,C 180,E1 -8736.34,E2 -8736.34} C_VEL
LIN {X 0,Y 445.722,Z 386.952,A -85,B 0,C 180,E1 -8737.93,E2 -8737.93} C_VEL
LIN {X 0,Y 446.015,Z 380.219,A -85,B 0,C 180,E1 -8739.295,E2 -8739.295} C_VEL
LIN {X 0,Y 446.421,Z 371.866,A -85,B 0,C 180,E1 -8740.66,E2 -8740.66} C_VEL
LIN {X 0,Y 446.974,Z 363.279,A -85,B 0,C 180,E1 -8741.795,E2 -8741.795} C_VEL
LIN {X 0,Y 447.515,Z 353.221,A -85,B 0,C 180,E1 -8742.879,E2 -8742.879} C_VEL
LIN {X 0,Y 448.064,Z 342.175,A -85,B 0,C 180,E1 -8743.84,E2 -8743.84} C_VEL
LIN {X 0,Y 448.681,Z 330.606,A -85,B 0,C 180,E1 -8744.63,E2 -8744.63} C_VEL
LIN {X 0,Y 449.28,Z 318.602,A -85,B 0,C 180,E1 -8745.248,E2 -8745.248} C_VEL
LIN {X 0,Y 449.724,Z 305.617,A -85,B 0,C 180,E1 -8745.726,E2 -8745.726} C_VEL
LIN {X 0,Y 450.073,Z 291.748,A -85,B 0,C 180,E1 -8746.033,E2 -8746.033} C_VEL
LIN {X 0,Y 450.626,Z 211.95,A -85,B 0,C 180,E1 -8747.326,E2 -8747.326} C_VEL
LIN {X 0,Y 447.375,Z 190.57,A -85,B 0,C 180,E1 -8747.813,E2 -8747.813} C_VEL
LIN {X 0,Y 448.327,Z 170.851,A -85,B 0,C 180,E1 -8751.375,E2 -8751.375} C_VEL
LIN {X 0,Y 449.039,Z 156.458,A -85,B 0,C 180,E1 -8754.013,E2 -8754.013} C_VEL
LIN {X 0,Y 446.864,Z 144.949,A -85,B 0,C 180,E1 -8756.302,E2 -8756.302} C_VEL
LIN {X 0,Y 446.45,Z 142.875,A -85,B 0,C 180,E1 -8756.732,E2 -8756.732} C_VEL
LIN {X 0,Y 446.433,Z 142.878,A -85,B 0,C 180,E1 -8760.02,E2 -8760.02} C_VEL
LIN {X 0,Y 446.428,Z 142.878,A -85,B 0,C 180,E1 -8763.449,E2 -8763.449} C_VEL
LIN {X 0,Y 446.404,Z 142.875,A -85,B 0,C 180,E1 -8766.746,E2 -8766.746} C_VEL
LIN {X 0,Y 446.406,Z 142.881,A -85,B 0,C 180,E1 -8769.517,E2 -8769.517} C_VEL
LIN {X 0,Y 446.38,Z 142.878,A -85,B 0,C 180,E1 -8772.611,E2 -8772.611} C_VEL
LIN {X 0,Y 446.454,Z 142.874,A -85,B 0,C 180,E1 -8775.104,E2 -8775.104} C_VEL
LIN {X 0,Y 446.405,Z 142.876,A -85,B 0,C 180,E1 -8778.606,E2 -8778.606} C_VEL
LIN {X 0,Y 446.415,Z 142.874,A -85,B 0,C 180,E1 -8781.922,E2 -8781.922} C_VEL
LIN {X 0,Y 446.427,Z 142.875,A -85,B 0,C 180,E1 -8785.476,E2 -8785.476} C_VEL
LIN {X 0,Y 446.412,Z 142.878,A -85,B 0,C 180,E1 -8788.699,E2 -8788.699} C_VEL
LIN {X 0,Y 446.43,Z 142.871,A -85,B 0,C 180,E1 -8791.836,E2 -8791.836} C_VEL
LIN {X 0,Y 446.426,Z 142.88,A -85,B 0,C 180,E1 -8794.845,E2 -8794.845} C_VEL
LIN {X 0,Y 446.452,Z 142.871,A -85,B 0,C 180,E1 -8798.246,E2 -8798.246} C_VEL
LIN {X 0,Y 446.443,Z 142.87,A -85,B 0,C 180,E1 -8801.648,E2 -8801.648} C_VEL
LIN {X 0,Y 446.464,Z 142.873,A -85,B 0,C 180,E1 -8804.478,E2 -8804.478} C_VEL
LIN {X 0,Y 446.522,Z 142.86,A -85,B 0,C 180,E1 -8807.383,E2 -8807.383} C_VEL
LIN {X 0,Y 446.522,Z 142.862,A -85,B 0,C 180,E1 -8810.944,E2 -8810.944} C_VEL
LIN {X 0,Y 446.61,Z 142.85,A -85,B 0,C 180,E1 -8813.675,E2 -8813.675} C_VEL
LIN {X 0,Y 446.657,Z 142.843,A -85,B 0,C 180,E1 -8817.294,E2 -8817.294} C_VEL
LIN {X 0,Y 446.741,Z 142.837,A -85,B 0,C 180,E1 -8819.999,E2 -8819.999} C_VEL
LIN {X 0,Y 446.655,Z 142.845,A -85,B 0,C 180,E1 -8822.705,E2 -8822.705} C_VEL
LIN {X 0,Y 446.608,Z 142.854,A -85,B 0,C 180,E1 -8826.323,E2 -8826.323} C_VEL
LIN {X 0,Y 446.512,Z 142.861,A -85,B 0,C 180,E1 -8829.055,E2 -8829.055} C_VEL
LIN {X 0,Y 446.524,Z 142.86,A -85,B 0,C 180,E1 -8832.729,E2 -8832.729} C_VEL
LIN {X 0,Y 446.452,Z 142.872,A -85,B 0,C 180,E1 -8836.206,E2 -8836.206} C_VEL
LIN {X 0,Y 446.433,Z 142.873,A -85,B 0,C 180,E1 -8839.304,E2 -8839.304} C_VEL
LIN {X 0,Y 446.412,Z 142.876,A -85,B 0,C 180,E1 -8842.199,E2 -8842.199} C_VEL
LIN {X 0,Y 446.421,Z 142.875,A -85,B 0,C 180,E1 -8845.154,E2 -8845.154} C_VEL
LIN {X 0,Y 446.416,Z 142.874,A -85,B 0,C 180,E1 -8848.182,E2 -8848.182} C_VEL
LIN {X 0,Y 446.407,Z 142.88,A -85,B 0,C 180,E1 -8851.3,E2 -8851.3} C_VEL
LIN {X 0,Y 446.42,Z 142.873,A -85,B 0,C 180,E1 -8854.523,E2 -8854.523} C_VEL
LIN {X 0,Y 446.402,Z 142.875,A -85,B 0,C 180,E1 -8858.076,E2 -8858.076} C_VEL
LIN {X 0,Y 446.397,Z 142.881,A -85,B 0,C 180,E1 -8861.393,E2 -8861.393} C_VEL
LIN {X 0,Y 446.446,Z 142.877,A -85,B 0,C 180,E1 -8865.103,E2 -8865.103} C_VEL
LIN {X 0,Y 446.396,Z 142.878,A -85,B 0,C 180,E1 -8868.605,E2 -8868.605} C_VEL
LIN {X 0,Y 446.405,Z 142.875,A -85,B 0,C 180,E1 -8871.921,E2 -8871.921} C_VEL
LIN {X 0,Y 446.416,Z 142.875,A -85,B 0,C 180,E1 -8875.475,E2 -8875.475} C_VEL
LIN {X 0,Y 446.401,Z 142.881,A -85,B 0,C 180,E1 -8878.698,E2 -8878.698} C_VEL
LIN {X 0,Y 446.417,Z 142.873,A -85,B 0,C 180,E1 -8881.836,E2 -8881.836} C_VEL
LIN {X 0,Y 446.414,Z 142.879,A -85,B 0,C 180,E1 -8884.845,E2 -8884.845} C_VEL
LIN {X 0,Y 446.44,Z 142.874,A -85,B 0,C 180,E1 -8888.245,E2 -8888.245} C_VEL
LIN {X 0,Y 446.431,Z 142.871,A -85,B 0,C 180,E1 -8891.648,E2 -8891.648} C_VEL
LIN {X 0,Y 446.45,Z 142.876,A -85,B 0,C 180,E1 -8894.477,E2 -8894.477} C_VEL
LIN {X 0,Y 446.509,Z 142.862,A -85,B 0,C 180,E1 -8897.384,E2 -8897.384} C_VEL
LIN {X 0,Y 446.5,Z 142.863,A -85,B 0,C 180,E1 -8900.944,E2 -8900.944} C_VEL
LIN {X 0,Y 446.596,Z 142.852,A -85,B 0,C 180,E1 -8903.675,E2 -8903.675} C_VEL
LIN {X 0,Y 446.549,Z 142.86,A -85,B 0,C 180,E1 -8906.964,E2 -8906.964} C_VEL
LIN {X 0,Y 445.95,Z 142.936,A -85,B 0,C 180,E1 -8907.466,E2 -8907.466} C_VEL
LIN {X 0,Y 443.088,Z 143.296,A -85,B 0,C 180,E1 -8908.251,E2 -8908.251} C_VEL
LIN {X 0,Y 440.191,Z 143.654,A -85,B 0,C 180,E1 -8909.046,E2 -8909.046} C_VEL
LIN {X 0,Y 439.562,Z 143.732,A -85,B 0,C 180,E1 -8909.559,E2 -8909.559} C_VEL
LIN {X 0,Y 439.586,Z 143.758,A -85,B 0,C 180,E1 -8910.286,E2 -8910.286} C_VEL
LIN {X 0,Y 440.894,Z 152.5,A -85,B 0,C 180,E1 -8912.284,E2 -8912.284} C_VEL
LIN {X 0,Y 440.629,Z 160.291,A -85,B 0,C 180,E1 -8913.972,E2 -8913.972} C_VEL
LIN {X 0,Y 444.175,Z 178.003,A -85,B 0,C 180,E1 -8914.428,E2 -8914.428} C_VEL
LIN {X 0,Y 443.216,Z 267.572,A -85,B 0,C 180,E1 -8915.916,E2 -8915.916} C_VEL
LIN {X 0,Y 442.827,Z 280.881,A -85,B 0,C 180,E1 -8916.321,E2 -8916.321} C_VEL
LIN {X 0,Y 442.461,Z 293.525,A -85,B 0,C 180,E1 -8916.899,E2 -8916.899} C_VEL
LIN {X 0,Y 441.974,Z 305.601,A -85,B 0,C 180,E1 -8917.653,E2 -8917.653} C_VEL
LIN {X 0,Y 441.371,Z 316.97,A -85,B 0,C 180,E1 -8918.567,E2 -8918.567} C_VEL
LIN {X 0,Y 440.772,Z 327.592,A -85,B 0,C 180,E1 -8919.638,E2 -8919.638} C_VEL
LIN {X 0,Y 440.136,Z 336.957,A -85,B 0,C 180,E1 -8920.814,E2 -8920.814} C_VEL
LIN {X 0,Y 439.556,Z 345.684,A -85,B 0,C 180,E1 -8922.168,E2 -8922.168} C_VEL
LIN {X 0,Y 439.132,Z 353.326,A -85,B 0,C 180,E1 -8923.654,E2 -8923.654} C_VEL
LIN {X 0,Y 438.834,Z 358.257,A -85,B 0,C 180,E1 -8924.847,E2 -8924.847} C_VEL
LIN {X 0,Y 438.59,Z 363.113,A -85,B 0,C 180,E1 -8926.326,E2 -8926.326} C_VEL
LIN {X 0,Y 438.393,Z 366.588,A -85,B 0,C 180,E1 -8927.734,E2 -8927.734} C_VEL
LIN {X 0,Y 438.299,Z 368.682,A -85,B 0,C 180,E1 -8928.91,E2 -8928.91} C_VEL
LIN {X 0,Y 438.195,Z 370.591,A -85,B 0,C 180,E1 -8930.662,E2 -8930.662} C_VEL
LIN {X 0,Y 438.178,Z 371.001,A -85,B 0,C 180,E1 -8931.648,E2 -8931.648} C_VEL
LIN {X 0,Y 438.191,Z 370.984,A -85,B 0,C 180,E1 -8932.639,E2 -8932.639} C_VEL
LIN {X 0,Y 438.238,Z 370.257,A -85,B 0,C 180,E1 -8933.924,E2 -8933.924} C_VEL
LIN {X 0,Y 438.364,Z 368.079,A -85,B 0,C 180,E1 -8935.65,E2 -8935.65} C_VEL
LIN {X 0,Y 438.562,Z 364.915,A -85,B 0,C 180,E1 -8937.175,E2 -8937.175} C_VEL
LIN {X 0,Y 438.741,Z 360.404,A -85,B 0,C 180,E1 -8938.722,E2 -8938.722} C_VEL
LIN {X 0,Y 439.099,Z 354.739,A -85,B 0,C 180,E1 -8940.2,E2 -8940.2} C_VEL
LIN {X 0,Y 439.459,Z 348.061,A -85,B 0,C 180,E1 -8941.584,E2 -8941.584} C_VEL
LIN {X 0,Y 439.988,Z 340.237,A -85,B 0,C 180,E1 -8942.894,E2 -8942.894} C_VEL
LIN {X 0,Y 440.631,Z 330.416,A -85,B 0,C 180,E1 -8944.21,E2 -8944.21} C_VEL
LIN {X 0,Y 441.286,Z 319.821,A -85,B 0,C 180,E1 -8945.349,E2 -8945.349} C_VEL
LIN {X 0,Y 441.883,Z 310.108,A -85,B 0,C 180,E1 -8946.19,E2 -8946.19} C_VEL
LIN {X 0,Y 442.507,Z 298.626,A -85,B 0,C 180,E1 -8946.98,E2 -8946.98} C_VEL
LIN {X 0,Y 442.944,Z 286.026,A -85,B 0,C 180,E1 -8947.637,E2 -8947.637} C_VEL
LIN {X 0,Y 443.264,Z 273.045,A -85,B 0,C 180,E1 -8948.114,E2 -8948.114} C_VEL
LIN {X 0,Y 443.533,Z 258.566,A -85,B 0,C 180,E1 -8948.421,E2 -8948.421} C_VEL
LIN {X 0,Y 444.382,Z 177.666,A -85,B 0,C 180,E1 -8949.753,E2 -8949.753} C_VEL
LIN {X 0,Y 440.894,Z 160.549,A -85,B 0,C 180,E1 -8950.21,E2 -8950.21} C_VEL
LIN {X 0,Y 441.022,Z 152.113,A -85,B 0,C 180,E1 -8952.013,E2 -8952.013} C_VEL
LIN {X 0,Y 439.403,Z 143.754,A -85,B 0,C 180,E1 -8953.968,E2 -8953.968} C_VEL
LIN {X 0,Y 439.399,Z 143.751,A -85,B 0,C 180,E1 -8957.371,E2 -8957.371} C_VEL
LIN {X 0,Y 439.446,Z 143.747,A -85,B 0,C 180,E1 -8960.231,E2 -8960.231} C_VEL
LIN {X 0,Y 439.373,Z 143.761,A -85,B 0,C 180,E1 -8963.714,E2 -8963.714} C_VEL
LIN {X 0,Y 439.37,Z 143.755,A -85,B 0,C 180,E1 -8967.055,E2 -8967.055} C_VEL
LIN {X 0,Y 439.38,Z 143.749,A -85,B 0,C 180,E1 -8970.275,E2 -8970.275} C_VEL
LIN {X 0,Y 439.427,Z 143.751,A -85,B 0,C 180,E1 -8973.397,E2 -8973.397} C_VEL
LIN {X 0,Y 439.385,Z 143.75,A -85,B 0,C 180,E1 -8976.43,E2 -8976.43} C_VEL
LIN {X 0,Y 439.388,Z 143.754,A -85,B 0,C 180,E1 -8979.398,E2 -8979.398} C_VEL
LIN {X 0,Y 439.404,Z 143.747,A -85,B 0,C 180,E1 -8982.309,E2 -8982.309} C_VEL
LIN {X 0,Y 439.447,Z 143.745,A -85,B 0,C 180,E1 -8985.175,E2 -8985.175} C_VEL
LIN {X 0,Y 439.484,Z 143.737,A -85,B 0,C 180,E1 -8988.002,E2 -8988.002} C_VEL
LIN {X 0,Y 439.505,Z 143.731,A -85,B 0,C 180,E1 -8991.726,E2 -8991.726} C_VEL
LIN {X 0,Y 439.611,Z 143.725,A -85,B 0,C 180,E1 -8994.496,E2 -8994.496} C_VEL
LIN {X 0,Y 439.635,Z 143.72,A -85,B 0,C 180,E1 -8998.169,E2 -8998.169} C_VEL
LIN {X 0,Y 439.758,Z 143.702,A -85,B 0,C 180,E1 -9000.001,E2 -9000.001} C_VEL
LIN {X 0,Y 439.609,Z 143.722,A -85,B 0,C 180,E1 -9002.75,E2 -9002.75} C_VEL
LIN {X 0,Y 439.565,Z 143.726,A -85,B 0,C 180,E1 -9006.427,E2 -9006.427} C_VEL
LIN {X 0,Y 439.493,Z 143.735,A -85,B 0,C 180,E1 -9009.202,E2 -9009.202} C_VEL
LIN {X 0,Y 439.468,Z 143.739,A -85,B 0,C 180,E1 -9012.938,E2 -9012.938} C_VEL
LIN {X 0,Y 439.404,Z 143.745,A -85,B 0,C 180,E1 -9016.329,E2 -9016.329} C_VEL
LIN {X 0,Y 439.401,Z 143.754,A -85,B 0,C 180,E1 -9019.627,E2 -9019.627} C_VEL
LIN {X 0,Y 439.356,Z 143.752,A -85,B 0,C 180,E1 -9022.577,E2 -9022.577} C_VEL
LIN {X 0,Y 439.368,Z 143.753,A -85,B 0,C 180,E1 -9025.588,E2 -9025.588} C_VEL
LIN {X 0,Y 439.379,Z 143.751,A -85,B 0,C 180,E1 -9028.677,E2 -9028.677} C_VEL
LIN {X 0,Y 439.345,Z 143.756,A -85,B 0,C 180,E1 -9032.025,E2 -9032.025} C_VEL
LIN {X 0,Y 439.383,Z 143.754,A -85,B 0,C 180,E1 -9035.338,E2 -9035.338} C_VEL
LIN {X 0,Y 439.349,Z 143.754,A -85,B 0,C 180,E1 -9038.599,E2 -9038.599} C_VEL
LIN {X 0,Y 439.346,Z 143.757,A -85,B 0,C 180,E1 -9042.211,E2 -9042.211} C_VEL
LIN {X 0,Y 439.399,Z 143.755,A -85,B 0,C 180,E1 -9045.27,E2 -9045.27} C_VEL
LIN {X 0,Y 439.356,Z 143.76,A -85,B 0,C 180,E1 -9049.016,E2 -9049.016} C_VEL
LIN {X 0,Y 439.344,Z 143.759,A -85,B 0,C 180,E1 -9052.564,E2 -9052.564} C_VEL
LIN {X 0,Y 439.397,Z 143.753,A -85,B 0,C 180,E1 -9054.844,E2 -9054.844} C_VEL
LIN {X 0,Y 439.372,Z 143.755,A -85,B 0,C 180,E1 -9058.14,E2 -9058.14} C_VEL
LIN {X 0,Y 439.402,Z 143.751,A -85,B 0,C 180,E1 -9061.607,E2 -9061.607} C_VEL
LIN {X 0,Y 439.384,Z 143.806,A -85,B 0,C 180,E1 -9063.073,E2 -9063.073} C_VEL
LIN {X 0,Y 441.84,Z 156.062,A -85,B 0,C 180,E1 -9065.571,E2 -9065.571} C_VEL
LIN {X 0,Y 442.006,Z 160.021,A -85,B 0,C 180,E1 -9066.329,E2 -9066.329} C_VEL
LIN {X 0,Y 440.979,Z 178.193,A -85,B 0,C 180,E1 -9069.678,E2 -9069.678} C_VEL
LIN {X 0,Y 440.416,Z 189.884,A -85,B 0,C 180,E1 -9071.81,E2 -9071.81} C_VEL
LIN {X 0,Y 444.051,Z 213.619,A -85,B 0,C 180,E1 -9072.371,E2 -9072.371} C_VEL
LIN {X 0,Y 443.243,Z 298.987,A -85,B 0,C 180,E1 -9073.802,E2 -9073.802} C_VEL
LIN {X 0,Y 442.782,Z 312.042,A -85,B 0,C 180,E1 -9074.198,E2 -9074.198} C_VEL
LIN {X 0,Y 442.156,Z 325.217,A -85,B 0,C 180,E1 -9074.796,E2 -9074.796} C_VEL
LIN {X 0,Y 441.467,Z 337.905,A -85,B 0,C 180,E1 -9075.597,E2 -9075.597} C_VEL
LIN {X 0,Y 440.821,Z 349.45,A -85,B 0,C 180,E1 -9076.539,E2 -9076.539} C_VEL
LIN {X 0,Y 440.257,Z 359.39,A -85,B 0,C 180,E1 -9077.555,E2 -9077.555} C_VEL
LIN {X 0,Y 439.675,Z 368.573,A -85,B 0,C 180,E1 -9078.708,E2 -9078.708} C_VEL
LIN {X 0,Y 439.119,Z 377.531,A -85,B 0,C 180,E1 -9080.093,E2 -9080.093} C_VEL
LIN {X 0,Y 438.771,Z 384.745,A -85,B 0,C 180,E1 -9081.48,E2 -9081.48} C_VEL
LIN {X 0,Y 438.498,Z 391.32,A -85,B 0,C 180,E1 -9083.096,E2 -9083.096} C_VEL
LIN {X 0,Y 438.361,Z 395.673,A -85,B 0,C 180,E1 -9084.48,E2 -9084.48} C_VEL
LIN {X 0,Y 438.34,Z 397.981,A -85,B 0,C 180,E1 -9085.402,E2 -9085.402} C_VEL
LIN {X 0,Y 438.282,Z 399.846,A -85,B 0,C 180,E1 -9086.323,E2 -9086.323} C_VEL
LIN {X 0,Y 438.342,Z 401.248,A -85,B 0,C 180,E1 -9087.243,E2 -9087.243} C_VEL
LIN {X 0,Y 438.281,Z 402.859,A -85,B 0,C 180,E1 -9089.081,E2 -9089.081} C_VEL
LIN {X 0,Y 438.285,Z 403.07,A -85,B 0,C 180,E1 -9090,E2 -9090} C_VEL
LIN {X 0,Y 438.296,Z 402.234,A -85,B 0,C 180,E1 -9091.838,E2 -9091.838} C_VEL
LIN {X 0,Y 438.342,Z 401.231,A -85,B 0,C 180,E1 -9092.757,E2 -9092.757} C_VEL
LIN {X 0,Y 438.283,Z 399.813,A -85,B 0,C 180,E1 -9093.678,E2 -9093.678} C_VEL
LIN {X 0,Y 438.378,Z 396.853,A -85,B 0,C 180,E1 -9095.059,E2 -9095.059} C_VEL
LIN {X 0,Y 438.426,Z 392.839,A -85,B 0,C 180,E1 -9096.443,E2 -9096.443} C_VEL
LIN {X 0,Y 438.666,Z 386.662,A -85,B 0,C 180,E1 -9098.059,E2 -9098.059} C_VEL
LIN {X 0,Y 438.958,Z 379.92,A -85,B 0,C 180,E1 -9099.446,E2 -9099.446} C_VEL
LIN {X 0,Y 439.392,Z 371.557,A -85,B 0,C 180,E1 -9100.833,E2 -9100.833} C_VEL
LIN {X 0,Y 440,Z 362.956,A -85,B 0,C 180,E1 -9101.985,E2 -9101.985} C_VEL
LIN {X 0,Y 440.523,Z 353.338,A -85,B 0,C 180,E1 -9103.042,E2 -9103.042} C_VEL
LIN {X 0,Y 441.137,Z 341.818,A -85,B 0,C 180,E1 -9104.061,E2 -9104.061} C_VEL
LIN {X 0,Y 441.805,Z 330.211,A -85,B 0,C 180,E1 -9104.863,E2 -9104.863} C_VEL
LIN {X 0,Y 442.426,Z 318.158,A -85,B 0,C 180,E1 -9105.49,E2 -9105.49} C_VEL
LIN {X 0,Y 442.907,Z 305.095,A -85,B 0,C 180,E1 -9105.975,E2 -9105.975} C_VEL
LIN {X 0,Y 443.239,Z 292.741,A -85,B 0,C 180,E1 -9106.258,E2 -9106.258} C_VEL
LIN {X 0,Y 443.91,Z 213.35,A -85,B 0,C 180,E1 -9107.561,E2 -9107.561} C_VEL
LIN {X 0,Y 440.403,Z 190.212,A -85,B 0,C 180,E1 -9108.116,E2 -9108.116} C_VEL
LIN {X 0,Y 441.471,Z 170.553,A -85,B 0,C 180,E1 -9111.724,E2 -9111.724} C_VEL
LIN {X 0,Y 442.077,Z 157.471,A -85,B 0,C 180,E1 -9114.165,E2 -9114.165} C_VEL
LIN {X 0,Y 439.419,Z 143.751,A -85,B 0,C 180,E1 -9116.958,E2 -9116.958} C_VEL
LIN {X 0,Y 439.383,Z 143.755,A -85,B 0,C 180,E1 -9120.26,E2 -9120.26} C_VEL
LIN {X 0,Y 439.368,Z 143.757,A -85,B 0,C 180,E1 -9123.717,E2 -9123.717} C_VEL
LIN {X 0,Y 439.376,Z 143.751,A -85,B 0,C 180,E1 -9126.287,E2 -9126.287} C_VEL
LIN {X 0,Y 439.363,Z 143.755,A -85,B 0,C 180,E1 -9129.78,E2 -9129.78} C_VEL
LIN {X 0,Y 439.337,Z 143.755,A -85,B 0,C 180,E1 -9132.62,E2 -9132.62} C_VEL
LIN {X 0,Y 439.401,Z 143.754,A -85,B 0,C 180,E1 -9135.27,E2 -9135.27} C_VEL
LIN {X 0,Y 439.358,Z 143.757,A -85,B 0,C 180,E1 -9139.016,E2 -9139.016} C_VEL
LIN {X 0,Y 439.372,Z 143.753,A -85,B 0,C 180,E1 -9141.609,E2 -9141.609} C_VEL
LIN {X 0,Y 439.4,Z 143.752,A -85,B 0,C 180,E1 -9144.843,E2 -9144.843} C_VEL
LIN {X 0,Y 439.371,Z 143.751,A -85,B 0,C 180,E1 -9148.139,E2 -9148.139} C_VEL
LIN {X 0,Y 439.405,Z 143.747,A -85,B 0,C 180,E1 -9151.606,E2 -9151.606} C_VEL
LIN {X 0,Y 439.371,Z 143.753,A -85,B 0,C 180,E1 -9154.412,E2 -9154.412} C_VEL
LIN {X 0,Y 439.365,Z 143.752,A -85,B 0,C 180,E1 -9157.424,E2 -9157.424} C_VEL
LIN {X 0,Y 439.446,Z 143.749,A -85,B 0,C 180,E1 -9160.663,E2 -9160.663} C_VEL
LIN {X 0,Y 439.424,Z 143.747,A -85,B 0,C 180,E1 -9164.222,E2 -9164.222} C_VEL
LIN {X 0,Y 439.49,Z 143.736,A -85,B 0,C 180,E1 -9167.285,E2 -9167.285} C_VEL
LIN {X 0,Y 439.488,Z 143.74,A -85,B 0,C 180,E1 -9170.797,E2 -9170.797} C_VEL
LIN {X 0,Y 439.563,Z 143.727,A -85,B 0,C 180,E1 -9173.573,E2 -9173.573} C_VEL
LIN {X 0,Y 439.41,Z 143.746,A -85,B 0,C 180,E1 -9175.412,E2 -9175.412} C_VEL
LIN {X 0,Y 439.631,Z 143.725,A -85,B 0,C 180,E1 -9178.167,E2 -9178.167} C_VEL
LIN {X 0,Y 439.692,Z 143.716,A -85,B 0,C 180,E1 -9179.999,E2 -9179.999} C_VEL
LIN {X 0,Y 439.607,Z 143.723,A -85,B 0,C 180,E1 -9182.748,E2 -9182.748} C_VEL
LIN {X 0,Y 439.561,Z 143.73,A -85,B 0,C 180,E1 -9186.425,E2 -9186.425} C_VEL
LIN {X 0,Y 439.478,Z 143.738,A -85,B 0,C 180,E1 -9189.201,E2 -9189.201} C_VEL
LIN {X 0,Y 439.467,Z 143.739,A -85,B 0,C 180,E1 -9192.937,E2 -9192.937} C_VEL
LIN {X 0,Y 439.398,Z 143.749,A -85,B 0,C 180,E1 -9196.325,E2 -9196.325} C_VEL
LIN {X 0,Y 439.378,Z 143.756,A -85,B 0,C 180,E1 -9199.626,E2 -9199.626} C_VEL
LIN {X 0,Y 439.359,Z 143.752,A -85,B 0,C 180,E1 -9202.575,E2 -9202.575} C_VEL
LIN {X 0,Y 439.367,Z 143.759,A -85,B 0,C 180,E1 -9205.586,E2 -9205.586} C_VEL
LIN {X 0,Y 439.379,Z 143.75,A -85,B 0,C 180,E1 -9208.675,E2 -9208.675} C_VEL
LIN {X 0,Y 439.364,Z 143.753,A -85,B 0,C 180,E1 -9212.028,E2 -9212.028} C_VEL
LIN {X 0,Y 439.388,Z 143.756,A -85,B 0,C 180,E1 -9215.338,E2 -9215.338} C_VEL
LIN {X 0,Y 439.355,Z 143.753,A -85,B 0,C 180,E1 -9218.597,E2 -9218.597} C_VEL
LIN {X 0,Y 439.345,Z 143.754,A -85,B 0,C 180,E1 -9222.209,E2 -9222.209} C_VEL
LIN {X 0,Y 439.393,Z 143.754,A -85,B 0,C 180,E1 -9225.269,E2 -9225.269} C_VEL
LIN {X 0,Y 439.349,Z 143.761,A -85,B 0,C 180,E1 -9229.015,E2 -9229.015} C_VEL
LIN {X 0,Y 439.362,Z 143.753,A -85,B 0,C 180,E1 -9231.608,E2 -9231.608} C_VEL
LIN {X 0,Y 439.389,Z 143.755,A -85,B 0,C 180,E1 -9234.843,E2 -9234.843} C_VEL
LIN {X 0,Y 439.36,Z 143.753,A -85,B 0,C 180,E1 -9238.138,E2 -9238.138} C_VEL
LIN {X 0,Y 439.38,Z 143.75,A -85,B 0,C 180,E1 -9241.609,E2 -9241.609} C_VEL
LIN {X 0,Y 439.36,Z 143.757,A -85,B 0,C 180,E1 -9244.412,E2 -9244.412} C_VEL
LIN {X 0,Y 439.353,Z 143.753,A -85,B 0,C 180,E1 -9247.424,E2 -9247.424} C_VEL
LIN {X 0,Y 439.434,Z 143.749,A -85,B 0,C 180,E1 -9250.663,E2 -9250.663} C_VEL
LIN {X 0,Y 439.409,Z 143.751,A -85,B 0,C 180,E1 -9254.222,E2 -9254.222} C_VEL
LIN {X 0,Y 439.477,Z 143.738,A -85,B 0,C 180,E1 -9257.285,E2 -9257.285} C_VEL
LIN {X 0,Y 439.467,Z 143.741,A -85,B 0,C 180,E1 -9260.797,E2 -9260.797} C_VEL
LIN {X 0,Y 439.549,Z 143.73,A -85,B 0,C 180,E1 -9263.574,E2 -9263.574} C_VEL
LIN {X 0,Y 439.397,Z 143.748,A -85,B 0,C 180,E1 -9265.413,E2 -9265.413} C_VEL
LIN {X 0,Y 439.618,Z 143.727,A -85,B 0,C 180,E1 -9268.168,E2 -9268.168} C_VEL
LIN {X 0,Y 439.562,Z 143.732,A -85,B 0,C 180,E1 -9269.559,E2 -9269.559} C_VEL
LIN {X 0,Y 439.378,Z 144.266,A -85,B 0,C 180,E1 -9270.066,E2 -9270.066} C_VEL
LIN {X 0,Y 438.348,Z 146.51,A -85,B 0,C 180,E1 -9270.776,E2 -9270.776} C_VEL
LIN {X 0,Y 434.113,Z 156.129,A -85,B 0,C 180,E1 -9272.732,E2 -9272.732} C_VEL
LIN {X 0,Y 433.804,Z 158.244,A -85,B 0,C 180,E1 -9273.183,E2 -9273.183} C_VEL
LIN {X 0,Y 433.733,Z 160.551,A -85,B 0,C 180,E1 -9273.687,E2 -9273.687} C_VEL
LIN {X 0,Y 437.405,Z 178.725,A -85,B 0,C 180,E1 -9274.163,E2 -9274.163} C_VEL
LIN {X 0,Y 436.417,Z 267.568,A -85,B 0,C 180,E1 -9275.66,E2 -9275.66} C_VEL
LIN {X 0,Y 436.033,Z 280.199,A -85,B 0,C 180,E1 -9276.043,E2 -9276.043} C_VEL
LIN {X 0,Y 435.601,Z 293.673,A -85,B 0,C 180,E1 -9276.659,E2 -9276.659} C_VEL
LIN {X 0,Y 435.093,Z 305.779,A -85,B 0,C 180,E1 -9277.425,E2 -9277.425} C_VEL
LIN {X 0,Y 434.438,Z 317.377,A -85,B 0,C 180,E1 -9278.372,E2 -9278.372} C_VEL
LIN {X 0,Y 433.816,Z 327.807,A -85,B 0,C 180,E1 -9279.441,E2 -9279.441} C_VEL
LIN {X 0,Y 433.221,Z 336.345,A -85,B 0,C 180,E1 -9280.516,E2 -9280.516} C_VEL
LIN {X 0,Y 432.572,Z 345.587,A -85,B 0,C 180,E1 -9281.955,E2 -9281.955} C_VEL
LIN {X 0,Y 432.128,Z 353.015,A -85,B 0,C 180,E1 -9283.4,E2 -9283.4} C_VEL
LIN {X 0,Y 431.803,Z 358.031,A -85,B 0,C 180,E1 -9284.612,E2 -9284.612} C_VEL
LIN {X 0,Y 431.558,Z 362.949,A -85,B 0,C 180,E1 -9286.094,E2 -9286.094} C_VEL
LIN {X 0,Y 431.355,Z 366.575,A -85,B 0,C 180,E1 -9287.543,E2 -9287.543} C_VEL
LIN {X 0,Y 431.196,Z 369.203,A -85,B 0,C 180,E1 -9289.036,E2 -9289.036} C_VEL
LIN {X 0,Y 431.127,Z 370.335,A -85,B 0,C 180,E1 -9290.019,E2 -9290.019} C_VEL
LIN {X 0,Y 431.103,Z 371.266,A -85,B 0,C 180,E1 -9291.687,E2 -9291.687} C_VEL
LIN {X 0,Y 431.092,Z 371.114,A -85,B 0,C 180,E1 -9293.033,E2 -9293.033} C_VEL
LIN {X 0,Y 431.145,Z 370.401,A -85,B 0,C 180,E1 -9294.101,E2 -9294.101} C_VEL
LIN {X 0,Y 431.201,Z 369.322,A -85,B 0,C 180,E1 -9295.072,E2 -9295.072} C_VEL
LIN {X 0,Y 431.374,Z 367.164,A -85,B 0,C 180,E1 -9296.356,E2 -9296.356} C_VEL
LIN {X 0,Y 431.553,Z 364.166,A -85,B 0,C 180,E1 -9297.654,E2 -9297.654} C_VEL
LIN {X 0,Y 431.769,Z 359.33,A -85,B 0,C 180,E1 -9299.23,E2 -9299.23} C_VEL
LIN {X 0,Y 432.095,Z 354.511,A -85,B 0,C 180,E1 -9300.455,E2 -9300.455} C_VEL
LIN {X 0,Y 432.518,Z 347.645,A -85,B 0,C 180,E1 -9301.877,E2 -9301.877} C_VEL
LIN {X 0,Y 433.089,Z 339.632,A -85,B 0,C 180,E1 -9303.208,E2 -9303.208} C_VEL
LIN {X 0,Y 433.795,Z 329.604,A -85,B 0,C 180,E1 -9304.544,E2 -9304.544} C_VEL
LIN {X 0,Y 434.418,Z 319.609,A -85,B 0,C 180,E1 -9305.62,E2 -9305.62} C_VEL
LIN {X 0,Y 435.138,Z 308.185,A -85,B 0,C 180,E1 -9306.593,E2 -9306.593} C_VEL
LIN {X 0,Y 435.782,Z 296.696,A -85,B 0,C 180,E1 -9307.358,E2 -9307.358} C_VEL
LIN {X 0,Y 436.186,Z 284.203,A -85,B 0,C 180,E1 -9307.991,E2 -9307.991} C_VEL
LIN {X 0,Y 436.519,Z 271.509,A -85,B 0,C 180,E1 -9308.429,E2 -9308.429} C_VEL
LIN {X 0,Y 436.826,Z 253.414,A -85,B 0,C 180,E1 -9308.782,E2 -9308.782} C_VEL
LIN {X 0,Y 437.607,Z 178.247,A -85,B 0,C 180,E1 -9310.042,E2 -9310.042} C_VEL
LIN {X 0,Y 434.003,Z 160.788,A -85,B 0,C 180,E1 -9310.524,E2 -9310.524} C_VEL
LIN {X 0,Y 434.032,Z 153.145,A -85,B 0,C 180,E1 -9312.183,E2 -9312.183} C_VEL
LIN {X 0,Y 432.363,Z 144.63,A -85,B 0,C 180,E1 -9314.174,E2 -9314.174} C_VEL
LIN {X 0,Y 432.362,Z 144.626,A -85,B 0,C 180,E1 -9317.01,E2 -9317.01} C_VEL
LIN {X 0,Y 432.354,Z 144.635,A -85,B 0,C 180,E1 -9319.818,E2 -9319.818} C_VEL
LIN {X 0,Y 432.312,Z 144.637,A -85,B 0,C 180,E1 -9323.024,E2 -9323.024} C_VEL
LIN {X 0,Y 432.357,Z 144.629,A -85,B 0,C 180,E1 -9325.997,E2 -9325.997} C_VEL
LIN {X 0,Y 432.345,Z 144.633,A -85,B 0,C 180,E1 -9329.49,E2 -9329.49} C_VEL
LIN {X 0,Y 432.39,Z 144.625,A -85,B 0,C 180,E1 -9332.929,E2 -9332.929} C_VEL
LIN {X 0,Y 432.37,Z 144.624,A -85,B 0,C 180,E1 -9336.024,E2 -9336.024} C_VEL
LIN {X 0,Y 432.349,Z 144.63,A -85,B 0,C 180,E1 -9339.047,E2 -9339.047} C_VEL
LIN {X 0,Y 432.359,Z 144.624,A -85,B 0,C 180,E1 -9342.011,E2 -9342.011} C_VEL
LIN {X 0,Y 432.395,Z 144.627,A -85,B 0,C 180,E1 -9344.927,E2 -9344.927} C_VEL
LIN {X 0,Y 432.46,Z 144.612,A -85,B 0,C 180,E1 -9347.804,E2 -9347.804} C_VEL
LIN {X 0,Y 432.465,Z 144.608,A -85,B 0,C 180,E1 -9351.591,E2 -9351.591} C_VEL
LIN {X 0,Y 432.587,Z 144.601,A -85,B 0,C 180,E1 -9354.407,E2 -9354.407} C_VEL
LIN {X 0,Y 432.604,Z 144.595,A -85,B 0,C 180,E1 -9358.139,E2 -9358.139} C_VEL
LIN {X 0,Y 432.728,Z 144.578,A -85,B 0,C 180,E1 -9360.001,E2 -9360.001} C_VEL
LIN {X 0,Y 432.563,Z 144.6,A -85,B 0,C 180,E1 -9362.795,E2 -9362.795} C_VEL
LIN {X 0,Y 432.579,Z 144.592,A -85,B 0,C 180,E1 -9365.595,E2 -9365.595} C_VEL
LIN {X 0,Y 432.464,Z 144.614,A -85,B 0,C 180,E1 -9368.411,E2 -9368.411} C_VEL
LIN {X 0,Y 432.462,Z 144.614,A -85,B 0,C 180,E1 -9372.197,E2 -9372.197} C_VEL
LIN {X 0,Y 432.391,Z 144.619,A -85,B 0,C 180,E1 -9376.041,E2 -9376.041} C_VEL
LIN {X 0,Y 432.388,Z 144.626,A -85,B 0,C 180,E1 -9379.485,E2 -9379.485} C_VEL
LIN {X 0,Y 432.306,Z 144.631,A -85,B 0,C 180,E1 -9382.966,E2 -9382.966} C_VEL
LIN {X 0,Y 432.32,Z 144.627,A -85,B 0,C 180,E1 -9386.036,E2 -9386.036} C_VEL
LIN {X 0,Y 432.317,Z 144.635,A -85,B 0,C 180,E1 -9389.19,E2 -9389.19} C_VEL
LIN {X 0,Y 432.307,Z 144.632,A -85,B 0,C 180,E1 -9392.445,E2 -9392.445} C_VEL
LIN {X 0,Y 432.332,Z 144.631,A -85,B 0,C 180,E1 -9395.819,E2 -9395.819} C_VEL
LIN {X 0,Y 432.313,Z 144.631,A -85,B 0,C 180,E1 -9398.71,E2 -9398.71} C_VEL
LIN {X 0,Y 432.302,Z 144.635,A -85,B 0,C 180,E1 -9401.802,E2 -9401.802} C_VEL
LIN {X 0,Y 432.336,Z 144.63,A -85,B 0,C 180,E1 -9404.348,E2 -9404.348} C_VEL
LIN {X 0,Y 432.303,Z 144.64,A -85,B 0,C 180,E1 -9407.019,E2 -9407.019} C_VEL
LIN {X 0,Y 432.291,Z 144.637,A -85,B 0,C 180,E1 -9409.828,E2 -9409.828} C_VEL
LIN {X 0,Y 432.304,Z 144.631,A -85,B 0,C 180,E1 -9413.022,E2 -9413.022} C_VEL
LIN {X 0,Y 432.335,Z 144.63,A -85,B 0,C 180,E1 -9416.002,E2 -9416.002} C_VEL
LIN {X 0,Y 432.349,Z 144.63,A -85,B 0,C 180,E1 -9419.49,E2 -9419.49} C_VEL
LIN {X 0,Y 432.351,Z 144.751,A -85,B 0,C 180,E1 -9422.827,E2 -9422.827} C_VEL
LIN {X 0,Y 434.87,Z 157.176,A -85,B 0,C 180,E1 -9425.408,E2 -9425.408} C_VEL
LIN {X 0,Y 435.095,Z 161.13,A -85,B 0,C 180,E1 -9426.183,E2 -9426.183} C_VEL
LIN {X 0,Y 434.004,Z 179.465,A -85,B 0,C 180,E1 -9429.618,E2 -9429.618} C_VEL
LIN {X 0,Y 433.519,Z 189.571,A -85,B 0,C 180,E1 -9431.493,E2 -9431.493} C_VEL
LIN {X 0,Y 437.262,Z 213.976,A -85,B 0,C 180,E1 -9432.089,E2 -9432.089} C_VEL
LIN {X 0,Y 436.513,Z 297.899,A -85,B 0,C 180,E1 -9433.515,E2 -9433.515} C_VEL
LIN {X 0,Y 435.993,Z 311.222,A -85,B 0,C 180,E1 -9433.916,E2 -9433.916} C_VEL
LIN {X 0,Y 435.355,Z 323.988,A -85,B 0,C 180,E1 -9434.492,E2 -9434.492} C_VEL
LIN {X 0,Y 434.7,Z 336.149,A -85,B 0,C 180,E1 -9435.248,E2 -9435.248} C_VEL
LIN {X 0,Y 433.96,Z 347.687,A -85,B 0,C 180,E1 -9436.178,E2 -9436.178} C_VEL
LIN {X 0,Y 433.315,Z 358.142,A -85,B 0,C 180,E1 -9437.233,E2 -9437.233} C_VEL
LIN {X 0,Y 432.811,Z 366.681,A -85,B 0,C 180,E1 -9438.289,E2 -9438.289} C_VEL
LIN {X 0,Y 432.208,Z 374.559,A -85,B 0,C 180,E1 -9439.46,E2 -9439.46} C_VEL
LIN {X 0,Y 431.799,Z 382.263,A -85,B 0,C 180,E1 -9440.869,E2 -9440.869} C_VEL
LIN {X 0,Y 431.461,Z 389.38,A -85,B 0,C 180,E1 -9442.513,E2 -9442.513} C_VEL
LIN {X 0,Y 431.318,Z 393.43,A -85,B 0,C 180,E1 -9443.698,E2 -9443.698} C_VEL
LIN {X 0,Y 431.268,Z 397.733,A -85,B 0,C 180,E1 -9445.326,E2 -9445.326} C_VEL
LIN {X 0,Y 431.189,Z 399.595,A -85,B 0,C 180,E1 -9446.262,E2 -9446.262} C_VEL
LIN {X 0,Y 431.238,Z 400.995,A -85,B 0,C 180,E1 -9447.198,E2 -9447.198} C_VEL
LIN {X 0,Y 431.219,Z 401.994,A -85,B 0,C 180,E1 -9448.132,E2 -9448.132} C_VEL
LIN {X 0,Y 431.196,Z 402.603,A -85,B 0,C 180,E1 -9449.066,E2 -9449.066} C_VEL
LIN {X 0,Y 431.198,Z 402.811,A -85,B 0,C 180,E1 -9450,E2 -9450} C_VEL
LIN {X 0,Y 431.22,Z 401.97,A -85,B 0,C 180,E1 -9451.868,E2 -9451.868} C_VEL
LIN {X 0,Y 431.238,Z 400.964,A -85,B 0,C 180,E1 -9452.803,E2 -9452.803} C_VEL
LIN {X 0,Y 431.189,Z 399.542,A -85,B 0,C 180,E1 -9453.738,E2 -9453.738} C_VEL
LIN {X 0,Y 431.287,Z 396.578,A -85,B 0,C 180,E1 -9455.142,E2 -9455.142} C_VEL
LIN {X 0,Y 431.344,Z 392.557,A -85,B 0,C 180,E1 -9456.549,E2 -9456.549} C_VEL
LIN {X 0,Y 431.595,Z 386.368,A -85,B 0,C 180,E1 -9458.192,E2 -9458.192} C_VEL
LIN {X 0,Y 431.906,Z 379.617,A -85,B 0,C 180,E1 -9459.601,E2 -9459.601} C_VEL
LIN {X 0,Y 432.393,Z 371.242,A -85,B 0,C 180,E1 -9461.01,E2 -9461.01} C_VEL
LIN {X 0,Y 433.01,Z 362.621,A -85,B 0,C 180,E1 -9462.181,E2 -9462.181} C_VEL
LIN {X 0,Y 433.599,Z 352.519,A -85,B 0,C 180,E1 -9463.301,E2 -9463.301} C_VEL
LIN {X 0,Y 434.221,Z 341.442,A -85,B 0,C 180,E1 -9464.29,E2 -9464.29} C_VEL
LIN {X 0,Y 434.908,Z 329.787,A -85,B 0,C 180,E1 -9465.105,E2 -9465.105} C_VEL
LIN {X 0,Y 435.557,Z 317.683,A -85,B 0,C 180,E1 -9465.741,E2 -9465.741} C_VEL
LIN {X 0,Y 436.094,Z 304.537,A -85,B 0,C 180,E1 -9466.231,E2 -9466.231} C_VEL
LIN {X 0,Y 436.426,Z 291.904,A -85,B 0,C 180,E1 -9466.519,E2 -9466.519} C_VEL
LIN {X 0,Y 437.018,Z 213.256,A -85,B 0,C 180,E1 -9467.835,E2 -9467.835} C_VEL
LIN {X 0,Y 433.449,Z 190.083,A -85,B 0,C 180,E1 -9468.383,E2 -9468.383} C_VEL
LIN {X 0,Y 434.574,Z 170.254,A -85,B 0,C 180,E1 -9472.087,E2 -9472.087} C_VEL
LIN {X 0,Y 435.093,Z 158.473,A -85,B 0,C 180,E1 -9474.324,E2 -9474.324} C_VEL
LIN {X 0,Y 432.357,Z 144.63,A -85,B 0,C 180,E1 -9477.205,E2 -9477.205} C_VEL
LIN {X 0,Y 432.35,Z 144.631,A -85,B 0,C 180,E1 -9480.51,E2 -9480.51} C_VEL
LIN {X 0,Y 432.337,Z 144.63,A -85,B 0,C 180,E1 -9483.998,E2 -9483.998} C_VEL
LIN {X 0,Y 432.324,Z 144.632,A -85,B 0,C 180,E1 -9487.196,E2 -9487.196} C_VEL
LIN {X 0,Y 432.294,Z 144.633,A -85,B 0,C 180,E1 -9490.172,E2 -9490.172} C_VEL
LIN {X 0,Y 432.307,Z 144.635,A -85,B 0,C 180,E1 -9493.063,E2 -9493.063} C_VEL
LIN {X 0,Y 432.337,Z 144.63,A -85,B 0,C 180,E1 -9495.665,E2 -9495.665} C_VEL
LIN {X 0,Y 432.312,Z 144.63,A -85,B 0,C 180,E1 -9498.402,E2 -9498.402} C_VEL
LIN {X 0,Y 432.336,Z 144.628,A -85,B 0,C 180,E1 -9501.849,E2 -9501.849} C_VEL
LIN {X 0,Y 432.332,Z 144.632,A -85,B 0,C 180,E1 -9505.322,E2 -9505.322} C_VEL
LIN {X 0,Y 432.32,Z 144.633,A -85,B 0,C 180,E1 -9508.653,E2 -9508.653} C_VEL
LIN {X 0,Y 432.339,Z 144.627,A -85,B 0,C 180,E1 -9511.873,E2 -9511.873} C_VEL
LIN {X 0,Y 432.329,Z 144.633,A -85,B 0,C 180,E1 -9514.997,E2 -9514.997} C_VEL
LIN {X 0,Y 432.36,Z 144.625,A -85,B 0,C 180,E1 -9518.045,E2 -9518.045} C_VEL
LIN {X 0,Y 432.386,Z 144.624,A -85,B 0,C 180,E1 -9521.029,E2 -9521.029} C_VEL
LIN {X 0,Y 432.393,Z 144.621,A -85,B 0,C 180,E1 -9523.959,E2 -9523.959} C_VEL
LIN {X 0,Y 432.464,Z 144.612,A -85,B 0,C 180,E1 -9527.803,E2 -9527.803} C_VEL
LIN {X 0,Y 432.453,Z 144.613,A -85,B 0,C 180,E1 -9531.589,E2 -9531.589} C_VEL
LIN {X 0,Y 432.575,Z 144.605,A -85,B 0,C 180,E1 -9534.405,E2 -9534.405} C_VEL
LIN {X 0,Y 432.6,Z 144.6,A -85,B 0,C 180,E1 -9538.137,E2 -9538.137} C_VEL
LIN {X 0,Y 432.643,Z 144.594,A -85,B 0,C 180,E1 -9539.999,E2 -9539.999} C_VEL
LIN {X 0,Y 432.56,Z 144.6,A -85,B 0,C 180,E1 -9542.793,E2 -9542.793} C_VEL
LIN {X 0,Y 432.518,Z 144.607,A -85,B 0,C 180,E1 -9546.53,E2 -9546.53} C_VEL
LIN {X 0,Y 432.423,Z 144.617,A -85,B 0,C 180,E1 -9549.353,E2 -9549.353} C_VEL
LIN {X 0,Y 432.433,Z 144.615,A -85,B 0,C 180,E1 -9552.802,E2 -9552.802} C_VEL
LIN {X 0,Y 432.357,Z 144.626,A -85,B 0,C 180,E1 -9556.452,E2 -9556.452} C_VEL
LIN {X 0,Y 432.314,Z 144.635,A -85,B 0,C 180,E1 -9559.961,E2 -9559.961} C_VEL
LIN {X 0,Y 432.308,Z 144.631,A -85,B 0,C 180,E1 -9562.964,E2 -9562.964} C_VEL
LIN {X 0,Y 432.318,Z 144.632,A -85,B 0,C 180,E1 -9566.034,E2 -9566.034} C_VEL
LIN {X 0,Y 432.32,Z 144.633,A -85,B 0,C 180,E1 -9569.188,E2 -9569.188} C_VEL
LIN {X 0,Y 432.32,Z 144.629,A -85,B 0,C 180,E1 -9572.442,E2 -9572.442} C_VEL
LIN {X 0,Y 432.334,Z 144.63,A -85,B 0,C 180,E1 -9575.817,E2 -9575.817} C_VEL
LIN {X 0,Y 432.298,Z 144.639,A -85,B 0,C 180,E1 -9579.347,E2 -9579.347} C_VEL
LIN {X 0,Y 432.3,Z 144.633,A -85,B 0,C 180,E1 -9581.8,E2 -9581.8} C_VEL
LIN {X 0,Y 432.33,Z 144.628,A -85,B 0,C 180,E1 -9584.346,E2 -9584.346} C_VEL
LIN {X 0,Y 432.298,Z 144.639,A -85,B 0,C 180,E1 -9587.017,E2 -9587.017} C_VEL
LIN {X 0,Y 432.303,Z 144.632,A -85,B 0,C 180,E1 -9589.824,E2 -9589.824} C_VEL
LIN {X 0,Y 432.299,Z 144.638,A -85,B 0,C 180,E1 -9593.021,E2 -9593.021} C_VEL
LIN {X 0,Y 432.327,Z 144.628,A -85,B 0,C 180,E1 -9596.001,E2 -9596.001} C_VEL
LIN {X 0,Y 432.335,Z 144.628,A -85,B 0,C 180,E1 -9599.491,E2 -9599.491} C_VEL
LIN {X 0,Y 432.313,Z 144.63,A -85,B 0,C 180,E1 -9601.871,E2 -9601.871} C_VEL
LIN {X 0,Y 432.316,Z 144.633,A -85,B 0,C 180,E1 -9604.996,E2 -9604.996} C_VEL
LIN {X 0,Y 432.348,Z 144.627,A -85,B 0,C 180,E1 -9608.045,E2 -9608.045} C_VEL
LIN {X 0,Y 432.373,Z 144.624,A -85,B 0,C 180,E1 -9611.029,E2 -9611.029} C_VEL
LIN {X 0,Y 432.378,Z 144.624,A -85,B 0,C 180,E1 -9613.959,E2 -9613.959} C_VEL
LIN {X 0,Y 432.446,Z 144.615,A -85,B 0,C 180,E1 -9617.803,E2 -9617.803} C_VEL
LIN {X 0,Y 432.438,Z 144.615,A -85,B 0,C 180,E1 -9621.589,E2 -9621.589} C_VEL
LIN {X 0,Y 432.562,Z 144.604,A -85,B 0,C 180,E1 -9624.405,E2 -9624.405} C_VEL
LIN {X 0,Y 432.587,Z 144.603,A -85,B 0,C 180,E1 -9628.138,E2 -9628.138} C_VEL
LIN {X 0,Y 432.629,Z 144.777,A -85,B 0,C 180,E1 -9630.116,E2 -9630.116} C_VEL
LIN {X 0,Y 433.911,Z 153.268,A -85,B 0,C 180,E1 -9632.088,E2 -9632.088} C_VEL
LIN {X 0,Y 433.804,Z 158.244,A -85,B 0,C 180,E1 -9633.183,E2 -9633.183} C_VEL
LIN {X 0,Y 433.055,Z 159.856,A -85,B 0,C 180,E1 -9633.403,E2 -9633.403} C_VEL
LIN {X 0,Y 430.735,Z 162.499,A -85,B 0,C 180,E1 -9633.538,E2 -9633.538} C_VEL
LIN {X 0,Y 427.53,Z 165.761,A -85,B 0,C 180,E1 -9633.518,E2 -9633.518} C_VEL
LIN {X 0,Y 424.772,Z 169.597,A -85,B 0,C 180,E1 -9633.464,E2 -9633.464} C_VEL
LIN {X 0,Y 424.033,Z 172.4,A -85,B 0,C 180,E1 -9633.479,E2 -9633.479} C_VEL
LIN {X 0,Y 424.431,Z 175.271,A -85,B 0,C 180,E1 -9633.542,E2 -9633.542} C_VEL
LIN {X 0,Y 425.853,Z 178.477,A -85,B 0,C 180,E1 -9633.66,E2 -9633.66} C_VEL
LIN {X 0,Y 429.918,Z 185.697,A -85,B 0,C 180,E1 -9633.969,E2 -9633.969} C_VEL
LIN {X 0,Y 430.563,Z 189.173,A -85,B 0,C 180,E1 -9634.059,E2 -9634.059} C_VEL
LIN {X 0,Y 429.567,Z 268.669,A -85,B 0,C 180,E1 -9635.427,E2 -9635.427} C_VEL
LIN {X 0,Y 429.14,Z 281.795,A -85,B 0,C 180,E1 -9635.845,E2 -9635.845} C_VEL
LIN {X 0,Y 428.749,Z 293.776,A -85,B 0,C 180,E1 -9636.411,E2 -9636.411} C_VEL
LIN {X 0,Y 428.226,Z 305.924,A -85,B 0,C 180,E1 -9637.189,E2 -9637.189} C_VEL
LIN {X 0,Y 427.547,Z 317.544,A -85,B 0,C 180,E1 -9638.151,E2 -9638.151} C_VEL
LIN {X 0,Y 426.933,Z 327.35,A -85,B 0,C 180,E1 -9639.164,E2 -9639.164} C_VEL
LIN {X 0,Y 426.327,Z 335.663,A -85,B 0,C 180,E1 -9640.207,E2 -9640.207} C_VEL
LIN {X 0,Y 425.739,Z 343.709,A -85,B 0,C 180,E1 -9641.425,E2 -9641.425} C_VEL
LIN {X 0,Y 425.239,Z 351.166,A -85,B 0,C 180,E1 -9642.817,E2 -9642.817} C_VEL
LIN {X 0,Y 424.799,Z 357.797,A -85,B 0,C 180,E1 -9644.369,E2 -9644.369} C_VEL
LIN {X 0,Y 424.528,Z 362.53,A -85,B 0,C 180,E1 -9645.778,E2 -9645.778} C_VEL
LIN {X 0,Y 424.296,Z 366.541,A -85,B 0,C 180,E1 -9647.346,E2 -9647.346} C_VEL
LIN {X 0,Y 424.174,Z 368.475,A -85,B 0,C 180,E1 -9648.349,E2 -9648.349} C_VEL
LIN {X 0,Y 424.086,Z 369.905,A -85,B 0,C 180,E1 -9649.356,E2 -9649.356} C_VEL
LIN {X 0,Y 424.033,Z 370.911,A -85,B 0,C 180,E1 -9650.368,E2 -9650.368} C_VEL
LIN {X 0,Y 424.004,Z 371.553,A -85,B 0,C 180,E1 -9651.844,E2 -9651.844} C_VEL
LIN {X 0,Y 424.025,Z 371.185,A -85,B 0,C 180,E1 -9653.44,E2 -9653.44} C_VEL
LIN {X 0,Y 424.061,Z 370.352,A -85,B 0,C 180,E1 -9654.477,E2 -9654.477} C_VEL
LIN {X 0,Y 424.151,Z 369.005,A -85,B 0,C 180,E1 -9655.519,E2 -9655.519} C_VEL
LIN {X 0,Y 424.383,Z 366.045,A -85,B 0,C 180,E1 -9657.091,E2 -9657.091} C_VEL
LIN {X 0,Y 424.61,Z 361.787,A -85,B 0,C 180,E1 -9658.691,E2 -9658.691} C_VEL
LIN {X 0,Y 424.988,Z 356.321,A -85,B 0,C 180,E1 -9660.235,E2 -9660.235} C_VEL
LIN {X 0,Y 425.373,Z 350.011,A -85,B 0,C 180,E1 -9661.639,E2 -9661.639} C_VEL
LIN {X 0,Y 425.938,Z 342.493,A -85,B 0,C 180,E1 -9662.991,E2 -9662.991} C_VEL
LIN {X 0,Y 426.617,Z 333.352,A -85,B 0,C 180,E1 -9664.324,E2 -9664.324} C_VEL
LIN {X 0,Y 427.282,Z 323.947,A -85,B 0,C 180,E1 -9665.436,E2 -9665.436} C_VEL
LIN {X 0,Y 428.008,Z 313.494,A -85,B 0,C 180,E1 -9666.431,E2 -9666.431} C_VEL
LIN {X 0,Y 428.724,Z 301.42,A -85,B 0,C 180,E1 -9667.339,E2 -9667.339} C_VEL
LIN {X 0,Y 429.263,Z 289.111,A -85,B 0,C 180,E1 -9668.045,E2 -9668.045} C_VEL
LIN {X 0,Y 429.629,Z 275.752,A -85,B 0,C 180,E1 -9668.584,E2 -9668.584} C_VEL
LIN {X 0,Y 429.961,Z 261.884,A -85,B 0,C 180,E1 -9668.924,E2 -9668.924} C_VEL
LIN {X 0,Y 430.856,Z 178.941,A -85,B 0,C 180,E1 -9670.337,E2 -9670.337} C_VEL
LIN {X 0,Y 427.107,Z 161.066,A -85,B 0,C 180,E1 -9670.838,E2 -9670.838} C_VEL
LIN {X 0,Y 427.13,Z 154.758,A -85,B 0,C 180,E1 -9672.233,E2 -9672.233} C_VEL
LIN {X 0,Y 425.345,Z 145.505,A -85,B 0,C 180,E1 -9674.449,E2 -9674.449} C_VEL
LIN {X 0,Y 425.34,Z 145.505,A -85,B 0,C 180,E1 -9678.034,E2 -9678.034} C_VEL
LIN {X 0,Y 425.318,Z 145.505,A -85,B 0,C 180,E1 -9681.105,E2 -9681.105} C_VEL
LIN {X 0,Y 425.296,Z 145.507,A -85,B 0,C 180,E1 -9684.665,E2 -9684.665} C_VEL
LIN {X 0,Y 425.262,Z 145.511,A -85,B 0,C 180,E1 -9688.074,E2 -9688.074} C_VEL
LIN {X 0,Y 425.329,Z 145.507,A -85,B 0,C 180,E1 -9691.369,E2 -9691.369} C_VEL
LIN {X 0,Y 425.294,Z 145.508,A -85,B 0,C 180,E1 -9694.556,E2 -9694.556} C_VEL
LIN {X 0,Y 425.287,Z 145.51,A -85,B 0,C 180,E1 -9697.662,E2 -9697.662} C_VEL
LIN {X 0,Y 425.36,Z 145.501,A -85,B 0,C 180,E1 -9700.705,E2 -9700.705} C_VEL
LIN {X 0,Y 425.388,Z 145.494,A -85,B 0,C 180,E1 -9703.689,E2 -9703.689} C_VEL
LIN {X 0,Y 425.413,Z 145.49,A -85,B 0,C 180,E1 -9707.599,E2 -9707.599} C_VEL
LIN {X 0,Y 425.409,Z 145.487,A -85,B 0,C 180,E1 -9711.45,E2 -9711.45} C_VEL
LIN {X 0,Y 425.542,Z 145.477,A -85,B 0,C 180,E1 -9714.314,E2 -9714.314} C_VEL
LIN {X 0,Y 425.573,Z 145.471,A -85,B 0,C 180,E1 -9718.108,E2 -9718.108} C_VEL
LIN {X 0,Y 425.697,Z 145.454,A -85,B 0,C 180,E1 -9720.001,E2 -9720.001} C_VEL
LIN {X 0,Y 425.518,Z 145.477,A -85,B 0,C 180,E1 -9722.841,E2 -9722.841} C_VEL
LIN {X 0,Y 425.533,Z 145.47,A -85,B 0,C 180,E1 -9725.688,E2 -9725.688} C_VEL
LIN {X 0,Y 425.409,Z 145.492,A -85,B 0,C 180,E1 -9728.551,E2 -9728.551} C_VEL
LIN {X 0,Y 425.415,Z 145.492,A -85,B 0,C 180,E1 -9732.402,E2 -9732.402} C_VEL
LIN {X 0,Y 425.307,Z 145.503,A -85,B 0,C 180,E1 -9735.332,E2 -9735.332} C_VEL
LIN {X 0,Y 425.315,Z 145.505,A -85,B 0,C 180,E1 -9738.299,E2 -9738.299} C_VEL
LIN {X 0,Y 425.289,Z 145.504,A -85,B 0,C 180,E1 -9741.319,E2 -9741.319} C_VEL
LIN {X 0,Y 425.3,Z 145.504,A -85,B 0,C 180,E1 -9744.651,E2 -9744.651} C_VEL
LIN {X 0,Y 425.245,Z 145.515,A -85,B 0,C 180,E1 -9747.566,E2 -9747.566} C_VEL
LIN {X 0,Y 425.286,Z 145.502,A -85,B 0,C 180,E1 -9750.76,E2 -9750.76} C_VEL
LIN {X 0,Y 425.289,Z 145.502,A -85,B 0,C 180,E1 -9754.283,E2 -9754.283} C_VEL
LIN {X 0,Y 425.269,Z 145.507,A -85,B 0,C 180,E1 -9757.696,E2 -9757.696} C_VEL
LIN {X 0,Y 425.247,Z 145.516,A -85,B 0,C 180,E1 -9761.383,E2 -9761.383} C_VEL
LIN {X 0,Y 425.287,Z 145.511,A -85,B 0,C 180,E1 -9764.717,E2 -9764.717} C_VEL
LIN {X 0,Y 425.266,Z 145.514,A -85,B 0,C 180,E1 -9768.046,E2 -9768.046} C_VEL
LIN {X 0,Y 425.28,Z 145.512,A -85,B 0,C 180,E1 -9771.099,E2 -9771.099} C_VEL
LIN {X 0,Y 425.297,Z 145.511,A -85,B 0,C 180,E1 -9774.664,E2 -9774.664} C_VEL
LIN {X 0,Y 425.266,Z 145.513,A -85,B 0,C 180,E1 -9778.073,E2 -9778.073} C_VEL
LIN {X 0,Y 425.307,Z 145.508,A -85,B 0,C 180,E1 -9781.366,E2 -9781.366} C_VEL
LIN {X 0,Y 425.302,Z 145.611,A -85,B 0,C 180,E1 -9782.554,E2 -9782.554} C_VEL
LIN {X 0,Y 427.899,Z 158.289,A -85,B 0,C 180,E1 -9785.24,E2 -9785.24} C_VEL
LIN {X 0,Y 428.182,Z 162.245,A -85,B 0,C 180,E1 -9786.031,E2 -9786.031} C_VEL
LIN {X 0,Y 427.031,Z 180.737,A -85,B 0,C 180,E1 -9789.555,E2 -9789.555} C_VEL
LIN {X 0,Y 426.56,Z 189.319,A -85,B 0,C 180,E1 -9791.172,E2 -9791.172} C_VEL
LIN {X 0,Y 430.483,Z 214.41,A -85,B 0,C 180,E1 -9791.798,E2 -9791.798} C_VEL
LIN {X 0,Y 429.732,Z 297.997,A -85,B 0,C 180,E1 -9793.247,E2 -9793.247} C_VEL
LIN {X 0,Y 429.139,Z 311.191,A -85,B 0,C 180,E1 -9793.652,E2 -9793.652} C_VEL
LIN {X 0,Y 428.512,Z 323.896,A -85,B 0,C 180,E1 -9794.238,E2 -9794.238} C_VEL
LIN {X 0,Y 427.813,Z 336.004,A -85,B 0,C 180,E1 -9795.005,E2 -9795.005} C_VEL
LIN {X 0,Y 427.058,Z 347.301,A -85,B 0,C 180,E1 -9795.929,E2 -9795.929} C_VEL
LIN {X 0,Y 426.343,Z 357.956,A -85,B 0,C 180,E1 -9797.021,E2 -9797.021} C_VEL
LIN {X 0,Y 425.808,Z 366.478,A -85,B 0,C 180,E1 -9798.094,E2 -9798.094} C_VEL
LIN {X 0,Y 425.082,Z 375.716,A -85,B 0,C 180,E1 -9799.522,E2 -9799.522} C_VEL
LIN {X 0,Y 424.702,Z 383.161,A -85,B 0,C 180,E1 -9800.955,E2 -9800.955} C_VEL
LIN {X 0,Y 424.383,Z 389.143,A -85,B 0,C 180,E1 -9802.387,E2 -9802.387} C_VEL
LIN {X 0,Y 424.213,Z 393.637,A -85,B 0,C 180,E1 -9803.74,E2 -9803.74} C_VEL
LIN {X 0,Y 424.197,Z 397.489,A -85,B 0,C 180,E1 -9805.248,E2 -9805.248} C_VEL
LIN {X 0,Y 424.1,Z 399.345,A -85,B 0,C 180,E1 -9806.199,E2 -9806.199} C_VEL
LIN {X 0,Y 424.134,Z 400.743,A -85,B 0,C 180,E1 -9807.151,E2 -9807.151} C_VEL
LIN {X 0,Y 424.144,Z 401.741,A -85,B 0,C 180,E1 -9808.101,E2 -9808.101} C_VEL
LIN {X 0,Y 424.114,Z 402.348,A -85,B 0,C 180,E1 -9809.051,E2 -9809.051} C_VEL
LIN {X 0,Y 424.113,Z 402.551,A -85,B 0,C 180,E1 -9810,E2 -9810} C_VEL
LIN {X 0,Y 424.144,Z 401.705,A -85,B 0,C 180,E1 -9811.899,E2 -9811.899} C_VEL
LIN {X 0,Y 424.135,Z 400.695,A -85,B 0,C 180,E1 -9812.85,E2 -9812.85} C_VEL
LIN {X 0,Y 424.1,Z 399.268,A -85,B 0,C 180,E1 -9813.801,E2 -9813.801} C_VEL
LIN {X 0,Y 424.198,Z 396.298,A -85,B 0,C 180,E1 -9815.228,E2 -9815.228} C_VEL
LIN {X 0,Y 424.259,Z 392.27,A -85,B 0,C 180,E1 -9816.659,E2 -9816.659} C_VEL
LIN {X 0,Y 424.528,Z 386.07,A -85,B 0,C 180,E1 -9818.329,E2 -9818.329} C_VEL
LIN {X 0,Y 424.879,Z 379.31,A -85,B 0,C 180,E1 -9819.762,E2 -9819.762} C_VEL
LIN {X 0,Y 425.398,Z 370.922,A -85,B 0,C 180,E1 -9821.194,E2 -9821.194} C_VEL
LIN {X 0,Y 426.016,Z 362.282,A -85,B 0,C 180,E1 -9822.384,E2 -9822.384} C_VEL
LIN {X 0,Y 426.653,Z 351.994,A -85,B 0,C 180,E1 -9823.538,E2 -9823.538} C_VEL
LIN {X 0,Y 427.342,Z 341.058,A -85,B 0,C 180,E1 -9824.525,E2 -9824.525} C_VEL
LIN {X 0,Y 428.036,Z 329.346,A -85,B 0,C 180,E1 -9825.353,E2 -9825.353} C_VEL
LIN {X 0,Y 428.704,Z 317.18,A -85,B 0,C 180,E1 -9825.999,E2 -9825.999} C_VEL
LIN {X 0,Y 429.248,Z 303.93,A -85,B 0,C 180,E1 -9826.497,E2 -9826.497} C_VEL
LIN {X 0,Y 429.593,Z 290.967,A -85,B 0,C 180,E1 -9826.789,E2 -9826.789} C_VEL
LIN {X 0,Y 430.261,Z 214.22,A -85,B 0,C 180,E1 -9828.093,E2 -9828.093} C_VEL
LIN {X 0,Y 426.505,Z 189.778,A -85,B 0,C 180,E1 -9828.693,E2 -9828.693} C_VEL
LIN {X 0,Y 427.696,Z 170.068,A -85,B 0,C 180,E1 -9832.436,E2 -9832.436} C_VEL
LIN {X 0,Y 428.228,Z 160.786,A -85,B 0,C 180,E1 -9834.224,E2 -9834.224} C_VEL
LIN {X 0,Y 425.938,Z 148.508,A -85,B 0,C 180,E1 -9836.791,E2 -9836.791} C_VEL
LIN {X 0,Y 425.327,Z 145.506,A -85,B 0,C 180,E1 -9837.468,E2 -9837.468} C_VEL
LIN {X 0,Y 425.292,Z 145.51,A -85,B 0,C 180,E1 -9840.816,E2 -9840.816} C_VEL
LIN {X 0,Y 425.295,Z 145.505,A -85,B 0,C 180,E1 -9844.284,E2 -9844.284} C_VEL
LIN {X 0,Y 425.28,Z 145.511,A -85,B 0,C 180,E1 -9847.695,E2 -9847.695} C_VEL
LIN {X 0,Y 425.248,Z 145.51,A -85,B 0,C 180,E1 -9850.514,E2 -9850.514} C_VEL
LIN {X 0,Y 425.251,Z 145.517,A -85,B 0,C 180,E1 -9853.349,E2 -9853.349} C_VEL
LIN {X 0,Y 425.261,Z 145.509,A -85,B 0,C 180,E1 -9856.043,E2 -9856.043} C_VEL
LIN {X 0,Y 425.258,Z 145.513,A -85,B 0,C 180,E1 -9859.484,E2 -9859.484} C_VEL
LIN {X 0,Y 425.281,Z 145.507,A -85,B 0,C 180,E1 -9862.489,E2 -9862.489} C_VEL
LIN {X 0,Y 425.291,Z 145.505,A -85,B 0,C 180,E1 -9865.815,E2 -9865.815} C_VEL
LIN {X 0,Y 425.293,Z 145.509,A -85,B 0,C 180,E1 -9869.239,E2 -9869.239} C_VEL
LIN {X 0,Y 425.265,Z 145.51,A -85,B 0,C 180,E1 -9872.436,E2 -9872.436} C_VEL
LIN {X 0,Y 425.328,Z 145.5,A -85,B 0,C 180,E1 -9875.6,E2 -9875.6} C_VEL
LIN {X 0,Y 425.295,Z 145.511,A -85,B 0,C 180,E1 -9878.681,E2 -9878.681} C_VEL
LIN {X 0,Y 425.317,Z 145.501,A -85,B 0,C 180,E1 -9881.701,E2 -9881.701} C_VEL
LIN {X 0,Y 425.308,Z 145.509,A -85,B 0,C 180,E1 -9884.668,E2 -9884.668} C_VEL
LIN {X 0,Y 425.417,Z 145.489,A -85,B 0,C 180,E1 -9887.598,E2 -9887.598} C_VEL
LIN {X 0,Y 425.402,Z 145.491,A -85,B 0,C 180,E1 -9891.448,E2 -9891.448} C_VEL
LIN {X 0,Y 425.529,Z 145.482,A -85,B 0,C 180,E1 -9894.312,E2 -9894.312} C_VEL
LIN {X 0,Y 425.569,Z 145.475,A -85,B 0,C 180,E1 -9898.106,E2 -9898.106} C_VEL
LIN {X 0,Y 425.594,Z 145.472,A -85,B 0,C 180,E1 -9899.999,E2 -9899.999} C_VEL
LIN {X 0,Y 425.516,Z 145.478,A -85,B 0,C 180,E1 -9902.839,E2 -9902.839} C_VEL
LIN {X 0,Y 425.479,Z 145.483,A -85,B 0,C 180,E1 -9906.639,E2 -9906.639} C_VEL
LIN {X 0,Y 425.384,Z 145.495,A -85,B 0,C 180,E1 -9909.509,E2 -9909.509} C_VEL
LIN {X 0,Y 425.395,Z 145.492,A -85,B 0,C 180,E1 -9912.902,E2 -9912.902} C_VEL
LIN {X 0,Y 425.315,Z 145.502,A -85,B 0,C 180,E1 -9916.582,E2 -9916.582} C_VEL
LIN {X 0,Y 425.297,Z 145.51,A -85,B 0,C 180,E1 -9919.622,E2 -9919.622} C_VEL
LIN {X 0,Y 425.287,Z 145.506,A -85,B 0,C 180,E1 -9922.338,E2 -9922.338} C_VEL
LIN {X 0,Y 425.259,Z 145.514,A -85,B 0,C 180,E1 -9925.447,E2 -9925.447} C_VEL
LIN {X 0,Y 425.299,Z 145.505,A -85,B 0,C 180,E1 -9928.857,E2 -9928.857} C_VEL
LIN {X 0,Y 425.261,Z 145.511,A -85,B 0,C 180,E1 -9931.926,E2 -9931.926} C_VEL
LIN {X 0,Y 425.293,Z 145.512,A -85,B 0,C 180,E1 -9935.335,E2 -9935.335} C_VEL
LIN {X 0,Y 425.275,Z 145.51,A -85,B 0,C 180,E1 -9938.9,E2 -9938.9} C_VEL
LIN {X 0,Y 425.253,Z 145.511,A -85,B 0,C 180,E1 -9942.654,E2 -9942.654} C_VEL
LIN {X 0,Y 425.281,Z 145.512,A -85,B 0,C 180,E1 -9945.282,E2 -9945.282} C_VEL
LIN {X 0,Y 425.245,Z 145.513,A -85,B 0,C 180,E1 -9948.617,E2 -9948.617} C_VEL
LIN {X 0,Y 425.279,Z 145.512,A -85,B 0,C 180,E1 -9951.099,E2 -9951.099} C_VEL
LIN {X 0,Y 425.289,Z 145.509,A -85,B 0,C 180,E1 -9954.663,E2 -9954.663} C_VEL
LIN {X 0,Y 425.254,Z 145.51,A -85,B 0,C 180,E1 -9958.072,E2 -9958.072} C_VEL
LIN {X 0,Y 425.289,Z 145.506,A -85,B 0,C 180,E1 -9961.364,E2 -9961.364} C_VEL
LIN {X 0,Y 425.252,Z 145.516,A -85,B 0,C 180,E1 -9964.552,E2 -9964.552} C_VEL
LIN {X 0,Y 425.284,Z 145.506,A -85,B 0,C 180,E1 -9967.729,E2 -9967.729} C_VEL
LIN {X 0,Y 425.353,Z 145.502,A -85,B 0,C 180,E1 -9970.703,E2 -9970.703} C_VEL
LIN {X 0,Y 425.311,Z 145.503,A -85,B 0,C 180,E1 -9973.685,E2 -9973.685} C_VEL
LIN {X 0,Y 425.386,Z 145.494,A -85,B 0,C 180,E1 -9977.097,E2 -9977.097} C_VEL
LIN {X 0,Y 425.373,Z 145.499,A -85,B 0,C 180,E1 -9980.49,E2 -9980.49} C_VEL
LIN {X 0,Y 425.467,Z 145.483,A -85,B 0,C 180,E1 -9983.36,E2 -9983.36} C_VEL
LIN {X 0,Y 425.336,Z 145.499,A -85,B 0,C 180,E1 -9985.261,E2 -9985.261} C_VEL
LIN {X 0,Y 425.556,Z 145.479,A -85,B 0,C 180,E1 -9988.107,E2 -9988.107} C_VEL
LIN {X 0,Y 425.566,Z 145.557,A -85,B 0,C 180,E1 -9989.882,E2 -9989.882} C_VEL
LIN {X 0,Y 426.986,Z 155.079,A -85,B 0,C 180,E1 -9992.122,E2 -9992.122} C_VEL
LIN {X 0,Y 426.797,Z 160.789,A -85,B 0,C 180,E1 -9993.392,E2 -9993.392} C_VEL
LIN {X 0,Y 430.624,Z 179.465,A -85,B 0,C 180,E1 -9993.892,E2 -9993.892} C_VEL
LIN {X 0,Y 430.563,Z 189.173,A -85,B 0,C 180,E1 -9994.059,E2 -9994.059} C_VEL
LIN {X 0,Y 429.824,Z 195.014,A -85,B 0,C 180,E1 -9994.13,E2 -9994.13} C_VEL
LIN {X 0,Y 424.197,Z 214.017,A -85,B 0,C 180,E1 -9994.225,E2 -9994.225} C_VEL
LIN {X 0,Y 423.439,Z 219.858,A -85,B 0,C 180,E1 -9994.296,E2 -9994.296} C_VEL
LIN {X 0,Y 422.769,Z 268.588,A -85,B 0,C 180,E1 -9995.156,E2 -9995.156} C_VEL
LIN {X 0,Y 422.335,Z 281.812,A -85,B 0,C 180,E1 -9995.58,E2 -9995.58} C_VEL
LIN {X 0,Y 421.903,Z 293.875,A -85,B 0,C 180,E1 -9996.156,E2 -9996.156} C_VEL
LIN {X 0,Y 421.352,Z 306.07,A -85,B 0,C 180,E1 -9996.945,E2 -9996.945} C_VEL
LIN {X 0,Y 420.651,Z 317.706,A -85,B 0,C 180,E1 -9997.923,E2 -9997.923} C_VEL
LIN {X 0,Y 420.04,Z 327.063,A -85,B 0,C 180,E1 -9998.9,E2 -9998.9} C_VEL
LIN {X 0,Y 419.314,Z 336.746,A -85,B 0,C 180,E1 -10000.136,E2 -10000.136} C_VEL
LIN {X 0,Y 418.589,Z 346.016,A -85,B 0,C 180,E1 -10001.623,E2 -10001.623} C_VEL
LIN {X 0,Y 418.042,Z 353.758,A -85,B 0,C 180,E1 -10003.181,E2 -10003.181} C_VEL
LIN {X 0,Y 417.658,Z 359.409,A -85,B 0,C 180,E1 -10004.62,E2 -10004.62} C_VEL
LIN {X 0,Y 417.358,Z 364.48,A -85,B 0,C 180,E1 -10006.297,E2 -10006.297} C_VEL
LIN {X 0,Y 417.174,Z 367.561,A -85,B 0,C 180,E1 -10007.652,E2 -10007.652} C_VEL
LIN {X 0,Y 417.016,Z 370.148,A -85,B 0,C 180,E1 -10009.309,E2 -10009.309} C_VEL
LIN {X 0,Y 416.914,Z 371.425,A -85,B 0,C 180,E1 -10010.732,E2 -10010.732} C_VEL
LIN {X 0,Y 416.927,Z 371.841,A -85,B 0,C 180,E1 -10012.013,E2 -10012.013} C_VEL
LIN {X 0,Y 416.961,Z 371.189,A -85,B 0,C 180,E1 -10013.861,E2 -10013.861} C_VEL
LIN {X 0,Y 417.019,Z 370.165,A -85,B 0,C 180,E1 -10014.918,E2 -10014.918} C_VEL
LIN {X 0,Y 417.125,Z 368.674,A -85,B 0,C 180,E1 -10015.98,E2 -10015.98} C_VEL
LIN {X 0,Y 417.373,Z 365.397,A -85,B 0,C 180,E1 -10017.585,E2 -10017.585} C_VEL
LIN {X 0,Y 417.639,Z 360.787,A -85,B 0,C 180,E1 -10019.21,E2 -10019.21} C_VEL
LIN {X 0,Y 418.014,Z 355.506,A -85,B 0,C 180,E1 -10020.646,E2 -10020.646} C_VEL
LIN {X 0,Y 418.538,Z 348.222,A -85,B 0,C 180,E1 -10022.218,E2 -10022.218} C_VEL
LIN {X 0,Y 419.198,Z 340.235,A -85,B 0,C 180,E1 -10023.591,E2 -10023.591} C_VEL
LIN {X 0,Y 419.924,Z 330.717,A -85,B 0,C 180,E1 -10024.909,E2 -10024.909} C_VEL
LIN {X 0,Y 420.651,Z 320.238,A -85,B 0,C 180,E1 -10026.082,E2 -10026.082} C_VEL
LIN {X 0,Y 421.425,Z 309.363,A -85,B 0,C 180,E1 -10027.045,E2 -10027.045} C_VEL
LIN {X 0,Y 422.149,Z 297.412,A -85,B 0,C 180,E1 -10027.872,E2 -10027.872} C_VEL
LIN {X 0,Y 422.587,Z 285.622,A -85,B 0,C 180,E1 -10028.494,E2 -10028.494} C_VEL
LIN {X 0,Y 423,Z 272.482,A -85,B 0,C 180,E1 -10028.974,E2 -10028.974} C_VEL
LIN {X 0,Y 423.306,Z 255.328,A -85,B 0,C 180,E1 -10029.328,E2 -10029.328} C_VEL
LIN {X 0,Y 424.262,Z 180.501,A -85,B 0,C 180,E1 -10030.621,E2 -10030.621} C_VEL
LIN {X 0,Y 420.237,Z 161.259,A -85,B 0,C 180,E1 -10031.188,E2 -10031.188} C_VEL
LIN {X 0,Y 420.231,Z 156.328,A -85,B 0,C 180,E1 -10032.295,E2 -10032.295} C_VEL
LIN {X 0,Y 418.286,Z 146.384,A -85,B 0,C 180,E1 -10034.697,E2 -10034.697} C_VEL
LIN {X 0,Y 418.289,Z 146.385,A -85,B 0,C 180,E1 -10037.774,E2 -10037.774} C_VEL
LIN {X 0,Y 418.261,Z 146.387,A -85,B 0,C 180,E1 -10041.56,E2 -10041.56} C_VEL
LIN {X 0,Y 418.256,Z 146.387,A -85,B 0,C 180,E1 -10045.16,E2 -10045.16} C_VEL
LIN {X 0,Y 418.243,Z 146.39,A -85,B 0,C 180,E1 -10047.473,E2 -10047.473} C_VEL
LIN {X 0,Y 418.266,Z 146.381,A -85,B 0,C 180,E1 -10050.896,E2 -10050.896} C_VEL
LIN {X 0,Y 418.269,Z 146.384,A -85,B 0,C 180,E1 -10054.097,E2 -10054.097} C_VEL
LIN {X 0,Y 418.237,Z 146.393,A -85,B 0,C 180,E1 -10057.265,E2 -10057.265} C_VEL
LIN {X 0,Y 418.282,Z 146.38,A -85,B 0,C 180,E1 -10060.365,E2 -10060.365} C_VEL
LIN {X 0,Y 418.316,Z 146.377,A -85,B 0,C 180,E1 -10063.406,E2 -10063.406} C_VEL
LIN {X 0,Y 418.347,Z 146.371,A -85,B 0,C 180,E1 -10067,E2 -10067} C_VEL
LIN {X 0,Y 418.34,Z 146.373,A -85,B 0,C 180,E1 -10070.329,E2 -10070.329} C_VEL
LIN {X 0,Y 418.461,Z 146.357,A -85,B 0,C 180,E1 -10073.249,E2 -10073.249} C_VEL
LIN {X 0,Y 418.334,Z 146.366,A -85,B 0,C 180,E1 -10075.182,E2 -10075.182} C_VEL
LIN {X 0,Y 418.542,Z 146.346,A -85,B 0,C 180,E1 -10078.076,E2 -10078.076} C_VEL
LIN {X 0,Y 418.666,Z 146.329,A -85,B 0,C 180,E1 -10080.001,E2 -10080.001} C_VEL
LIN {X 0,Y 418.475,Z 146.354,A -85,B 0,C 180,E1 -10082.889,E2 -10082.889} C_VEL
LIN {X 0,Y 418.49,Z 146.347,A -85,B 0,C 180,E1 -10085.784,E2 -10085.784} C_VEL
LIN {X 0,Y 418.378,Z 146.366,A -85,B 0,C 180,E1 -10088.696,E2 -10088.696} C_VEL
LIN {X 0,Y 418.316,Z 146.367,A -85,B 0,C 180,E1 -10091.632,E2 -10091.632} C_VEL
LIN {X 0,Y 418.282,Z 146.378,A -85,B 0,C 180,E1 -10094.598,E2 -10094.598} C_VEL
LIN {X 0,Y 418.258,Z 146.381,A -85,B 0,C 180,E1 -10097.606,E2 -10097.606} C_VEL
LIN {X 0,Y 418.248,Z 146.379,A -85,B 0,C 180,E1 -10100.664,E2 -10100.664} C_VEL
LIN {X 0,Y 418.257,Z 146.387,A -85,B 0,C 180,E1 -10103.784,E2 -10103.784} C_VEL
LIN {X 0,Y 418.207,Z 146.385,A -85,B 0,C 180,E1 -10107.042,E2 -10107.042} C_VEL
LIN {X 0,Y 418.235,Z 146.38,A -85,B 0,C 180,E1 -10110.274,E2 -10110.274} C_VEL
LIN {X 0,Y 418.229,Z 146.385,A -85,B 0,C 180,E1 -10113.68,E2 -10113.68} C_VEL
LIN {X 0,Y 418.233,Z 146.388,A -85,B 0,C 180,E1 -10117.226,E2 -10117.226} C_VEL
LIN {X 0,Y 418.207,Z 146.393,A -85,B 0,C 180,E1 -10120.951,E2 -10120.951} C_VEL
LIN {X 0,Y 418.203,Z 146.39,A -85,B 0,C 180,E1 -10123.728,E2 -10123.728} C_VEL
LIN {X 0,Y 418.201,Z 146.396,A -85,B 0,C 180,E1 -10126.448,E2 -10126.448} C_VEL
LIN {X 0,Y 418.209,Z 146.394,A -85,B 0,C 180,E1 -10129.133,E2 -10129.133} C_VEL
LIN {X 0,Y 418.239,Z 146.385,A -85,B 0,C 180,E1 -10132.776,E2 -10132.776} C_VEL
LIN {X 0,Y 418.235,Z 146.386,A -85,B 0,C 180,E1 -10136.322,E2 -10136.322} C_VEL
LIN {X 0,Y 418.244,Z 146.388,A -85,B 0,C 180,E1 -10139.728,E2 -10139.728} C_VEL
LIN {X 0,Y 418.269,Z 146.53,A -85,B 0,C 180,E1 -10142.281,E2 -10142.281} C_VEL
LIN {X 0,Y 420.791,Z 158.768,A -85,B 0,C 180,E1 -10144.93,E2 -10144.93} C_VEL
LIN {X 0,Y 421.27,Z 163.36,A -85,B 0,C 180,E1 -10145.875,E2 -10145.875} C_VEL
LIN {X 0,Y 420.119,Z 180.408,A -85,B 0,C 180,E1 -10149.177,E2 -10149.177} C_VEL
LIN {X 0,Y 419.673,Z 189.055,A -85,B 0,C 180,E1 -10150.839,E2 -10150.839} C_VEL
LIN {X 0,Y 423.646,Z 214.266,A -85,B 0,C 180,E1 -10151.485,E2 -10151.485} C_VEL
LIN {X 0,Y 423.74,Z 229.567,A -85,B 0,C 180,E1 -10151.763,E2 -10151.763} C_VEL
LIN {X 0,Y 422.963,Z 298.086,A -85,B 0,C 180,E1 -10152.971,E2 -10152.971} C_VEL
LIN {X 0,Y 422.326,Z 311.16,A -85,B 0,C 180,E1 -10153.38,E2 -10153.38} C_VEL
LIN {X 0,Y 421.684,Z 323.803,A -85,B 0,C 180,E1 -10153.976,E2 -10153.976} C_VEL
LIN {X 0,Y 420.937,Z 335.859,A -85,B 0,C 180,E1 -10154.754,E2 -10154.754} C_VEL
LIN {X 0,Y 420.141,Z 347.379,A -85,B 0,C 180,E1 -10155.716,E2 -10155.716} C_VEL
LIN {X 0,Y 419.404,Z 357.773,A -85,B 0,C 180,E1 -10156.802,E2 -10156.802} C_VEL
LIN {X 0,Y 418.833,Z 366.281,A -85,B 0,C 180,E1 -10157.892,E2 -10157.892} C_VEL
LIN {X 0,Y 418.065,Z 375.505,A -85,B 0,C 180,E1 -10159.344,E2 -10159.344} C_VEL
LIN {X 0,Y 417.639,Z 382.941,A -85,B 0,C 180,E1 -10160.801,E2 -10160.801} C_VEL
LIN {X 0,Y 417.331,Z 388.916,A -85,B 0,C 180,E1 -10162.258,E2 -10162.258} C_VEL
LIN {X 0,Y 417.12,Z 393.804,A -85,B 0,C 180,E1 -10163.769,E2 -10163.769} C_VEL
